// Exit action
//--------------------------------------------------------------------------------------
	IF (me.StateMachine.intState <> me.StateMachine.intStateNext) THEN
		// state is going to change
		;
	END_IF
END_METHOD

{attribute 'object_name' := 'sta_BELTONLYBusy'}
METHOD PROTECTED sta_BELTONLYBusy : BOOL
VAR
	bReady: BOOL;
	iErrorNumber: INT;
END_VAR
// state implemetation

// Entry action
//--------------------------------------------------------------------------------------
	IF (me.StateMachine.intState <> me.StateMachine.intStateLastCycle) THEN
		// state changed since last cycle
		me.StateMachine.intStateLastCycle := me.StateMachine.intState;
		
		// Set Outputs
		p_fbIBH^.setBeltOn();
		p_fbIBH^.setSpeed(In_diSpeed_mm_min := SIf.Par.diSpeed_mm_min);
		THIS^.lastSifPar := SIf.Par;
	END_IF

	
// Cyclic action
//--------------------------------------------------------------------------------------

	// Simulation
	IF (CIf.SwCfg.bolSimulation) THEN
		;
	END_IF
	
	// check if parameters have changed
	IF (TC2_SYSTEM.MEMCMP(pBuf1:=ADR(SIf.Par), pBuf2:=ADR(THIS^.lastSifPar), n:=SIZEOF(SIf.Par)) <> 0) THEN
		p_fbIBH^.setSpeed(In_diSpeed_mm_min := SIf.Par.diSpeed_mm_min);
		THIS^.lastSifPar := SIf.Par;
	END_IF
	
	// check timeouts
	IF me.StateMachine.udiTimeInState_ms>SIf.Par.udiTimeoutBeltOnlyBusy_ms THEN
		iErrorNumber := 100*me.StateMachine.intState+In_iStatus;
		pfbAlarmCtrl^.setAlarm(CIf.Info.intCtrlId,INT_TO_UDINT(E_ALM_OVN.TimeoutError),iErrorNumber,ADR(SIf.Alm),E_AlmState.RST,CIf.Job.eMe_ActivAlmClass);
		me.StateMachine.intStateNext := Base_PLC.cSTA_ERROR;
	ELSIF me.StateMachine.udiTimeInState_ms>SIf.Par.udiTimeoutBeltOnlyReaction_ms THEN
		IF NOT In_bBeltOn OR NOT ((In_iStatus=2) OR (In_iStatus=6)) THEN
			iErrorNumber := 100*me.StateMachine.intState+In_iStatus;
			pfbAlarmCtrl^.setAlarm(CIf.Info.intCtrlId,INT_TO_UDINT(E_ALM_OVN.TimeoutError),iErrorNumber,ADR(SIf.Alm),E_AlmState.RST,CIf.Job.eMe_ActivAlmClass);
			me.StateMachine.intStateNext := Base_PLC.cSTA_ERROR;
		END_IF
	END_IF
	
	// Check if ready
	bReady := TRUE;
	IF NOT In_bBeltOn OR NOT (In_iStatus=2) OR (In_iStatus=6) THEN
		bReady := FALSE;
	END_IF
	IF (ABS(THIS^.In_diSpeed_mm_min - SIf.Par.diSpeed_mm_min) > ABS(SIf.Par.diSpeedBand1_mm_min)) THEN
		bReady := FALSE;
	END_IF
	
	// State Change Condition
	IF (me.StateMachine.intStateNext <> Base_PLC.cSTA_ERROR) THEN
		CASE me.intCmd OF
			// OFF
			Base_PLC.cCMD_OFF:
				me.StateMachine.intStateNext := Base_PLC.cSTA_OFFBusy;
		ELSE
			// DEFAULT
			IF bReady THEN
				me.StateMachine.intStateNext := OVN_CmdState.cSTA_BELTONLY;
			END_IF
		END_CASE
	END_IF


// Exit action
//--------------------------------------------------------------------------------------
	IF (me.StateMachine.intState <> me.StateMachine.intStateNext) THEN
		// state is going to change
		;
	END_IF
END_METHOD

{attribute 'object_name' := 'sta_ERROR'}
METHOD PROTECTED sta_ERROR : BOOL
// state implemetation

// Entry action
//--------------------------------------------------------------------------------------
	IF (me.StateMachine.intState <> me.StateMachine.intStateLastCycle) THEN
		// state changed since last cycle
		me.StateMachine.intStateHistory := me.StateMachine.intStateLastCycle; // -> possibillity to go back to state before error
		me.StateMachine.intStateLastCycle := me.StateMachine.intState;
	END_IF

	
// Cyclic action
//--------------------------------------------------------------------------------------	
	
	// Simulation
	IF (CIf.SwCfg.bolSimulation) THEN
		;
	END_IF
	
	// Mark all tracked item as trash
	fbTracker.markAllTrash();
	
	// auto continue after Connection Error
	IF (iLastCalledAlarmNr=E_ALM_OVN.ConnectionError AND SIf.Cfg.bAutoContinueAfterConnectionError) THEN
		IF THIS^.In_bDriverConnected THEN
			CIf.Job.bolAlmReset := TRUE;
			pfbAlarmCtrl^.setAlarm(CIf.Info.intCtrlId,INT_TO_UDINT(E_ALM_OVN.ConnectionError),UDINT_TO_DINT(THIS^.In_udiDriverErrorID),ADR(SIf.Alm),E_AlmState.CLR,CIf.Job.eMe_ActivAlmClass);
		END_IF
	END_IF
	
	// State Change Condition
	IF (CIf.Job.bolAlmReset = TRUE) THEN
		p_fbIBH^.setAckError();
		me.StateMachine.intStateNext := cSTA_ERRORQuit;
	END_IF


// Exit action
//--------------------------------------------------------------------------------------
	IF (me.StateMachine.intState <> me.StateMachine.intStateNext) THEN
		// state is going to change
		;
	END_IF
END_METHOD

{attribute 'object_name' := 'sta_ERRORQuit'}
METHOD PROTECTED sta_ERRORQuit : BOOL
// state implemetation

// Entry action
//--------------------------------------------------------------------------------------
	IF (me.StateMachine.intState <> me.StateMachine.intStateLastCycle) THEN
		// state changed since last cycle
		me.StateMachine.intStateLastCycle := me.StateMachine.intState;
	END_IF

	
// Cyclic action
//--------------------------------------------------------------------------------------	
	
	// Simulation
	IF (CIf.SwCfg.bolSimulation) THEN
		;
	END_IF
	
	// State Change Condition
	CASE me.StateMachine.intStateHistory OF
		// RUN
		Base_PLC.cSTA_RUN, Base_PLC.cSTA_RUNBusy:
			me.StateMachine.intStateNext := Base_PLC.cSTA_RUNBusy;
		// PON
		Base_PLC.cSTA_PON, Base_PLC.cSTA_PONBusy:
			me.StateMachine.intStateNext := Base_PLC.cSTA_PONBusy;
		// STOP
		Base_PLC.cSTA_STOP, Base_PLC.cSTA_STOPBusy:
			me.StateMachine.intStateNext := Base_PLC.cSTA_STOPBusy;
		// BELTONLY
		OVN_CmdState.cSTA_BELTONLY, OVN_CmdState.cSTA_BELTONLYBusy:
			me.StateMachine.intStateNext := OVN_CmdState.cSTA_BELTONLYBusy;
	ELSE
		// DEFAULT
		me.StateMachine.intStateNext := Base_PLC.cSTA_OFFBusy;
	END_CASE


// Exit action
//--------------------------------------------------------------------------------------
	IF (me.StateMachine.intState <> me.StateMachine.intStateNext) THEN
		// state is going to change
		
		// Reset iLastCalledAlarmNr
		iLastCalledAlarmNr := E_ALM_OVN.NONE;
	END_IF
END_METHOD

{attribute 'object_name' := 'sta_OFF'}
METHOD PROTECTED sta_OFF : BOOL
// state implemetation

// Entry action
//--------------------------------------------------------------------------------------
	IF (me.StateMachine.intState <> me.StateMachine.intStateLastCycle) THEN
		// state changed since last cycle
		me.StateMachine.intStateLastCycle := me.StateMachine.intState;
	END_IF

	
// Cyclic action
//--------------------------------------------------------------------------------------

	// Simulation
	IF (CIf.SwCfg.bolSimulation) THEN
		;
	END_IF
	
	IF NOT In_bOff OR NOT (In_iStatus=1 OR In_iStatus=6 OR In_iStatus=5) THEN
		pfbAlarmCtrl^.setAlarm(CIf.Info.intCtrlId,INT_TO_UDINT(E_ALM_OVN.WrongMode),0,ADR(SIf.Alm),E_AlmState.RST,CIf.Job.eMe_ActivAlmClass);
		me.StateMachine.intStateNext := Base_PLC.cSTA_ERROR;
	END_IF
	
	// State Change Condition
	IF (me.StateMachine.intStateNext <> Base_PLC.cSTA_ERROR) THEN
		CASE me.intCmd OF
			// RUN
			Base_PLC.cCMD_RUN:
				me.StateMachine.intStateNext := Base_PLC.cSTA_RUNBusy;
			// BELTONLY
			OVN_CmdState.cCMD_BELTONLY:
				me.StateMachine.intStateNext := OVN_CmdState.cSTA_BELTONLYBusy;
		ELSE
			// DEFAULT
			;
		END_CASE
	END_IF


// Exit action
//--------------------------------------------------------------------------------------
	IF (me.StateMachine.intState <> me.StateMachine.intStateNext) THEN
		// state is going to change
		;
	END_IF
END_METHOD

{attribute 'object_name' := 'sta_OFFBusy'}
METHOD PROTECTED sta_OFFBusy : BOOL
VAR
	bReady: BOOL;
	iErrorNumber: INT;
END_VAR
// state implemetation

// Entry action
//--------------------------------------------------------------------------------------
	IF (me.StateMachine.intState <> me.StateMachine.intStateLastCycle) THEN
		// state changed since last cycle
		me.StateMachine.intStateLastCycle := me.StateMachine.intState;
		
		// Set Outputs
		p_fbIBH^.setOff();
		
		// mark all tracked items as trash
		fbTracker.markAllTrash();
	END_IF

	
// Cyclic action
//--------------------------------------------------------------------------------------

	// Simulation
	IF (CIf.SwCfg.bolSimulation) THEN
		;
	END_IF
	
	// check timeouts
	IF me.StateMachine.udiTimeInState_ms>SIf.Par.udiTimeoutOffBusy_ms THEN
		iErrorNumber := 100*me.StateMachine.intState+In_iStatus;
		pfbAlarmCtrl^.setAlarm(CIf.Info.intCtrlId,INT_TO_UDINT(E_ALM_OVN.TimeoutError),iErrorNumber,ADR(SIf.Alm),E_AlmState.RST,CIf.Job.eMe_ActivAlmClass);
		me.StateMachine.intStateNext := Base_PLC.cSTA_ERROR;
	ELSIF me.StateMachine.udiTimeInState_ms>SIf.Par.udiTimeoutOffBusyReaction_ms THEN
		IF NOT In_bOff OR NOT ((In_iStatus=1) OR (In_iStatus=6)) THEN
			iErrorNumber := 100*me.StateMachine.intState+In_iStatus;
			pfbAlarmCtrl^.setAlarm(CIf.Info.intCtrlId,INT_TO_UDINT(E_ALM_OVN.TimeoutError),iErrorNumber,ADR(SIf.Alm),E_AlmState.RST,CIf.Job.eMe_ActivAlmClass);
			me.StateMachine.intStateNext := Base_PLC.cSTA_ERROR;
		END_IF
	END_IF
	
	// check if ready
	bReady := TRUE;
	IF NOT In_bOff OR NOT (In_iStatus=1) OR (In_iStatus=6) THEN
		bReady := FALSE;
	END_IF
	
	// State Change Condition
	IF (me.StateMachine.intStateNext <> Base_PLC.cSTA_ERROR) THEN
		IF bReady THEN
			me.StateMachine.intStateNext := Base_PLC.cCMD_OFF;
		END_IF
	END_IF


// Exit action
//--------------------------------------------------------------------------------------
	IF (me.StateMachine.intState <> me.StateMachine.intStateNext) THEN
		// state is going to change
		;
	END_IF
END_METHOD

{attribute 'object_name' := 'sta_PON'}
METHOD PROTECTED sta_PON : BOOL
// state implemetation

// Entry action
//--------------------------------------------------------------------------------------
	IF (me.StateMachine.intState <> me.StateMachine.intStateLastCycle) THEN
		// state changed since last cycle
		me.StateMachine.intStateLastCycle := me.StateMachine.intState;
	END_IF

	
// Cyclic action
//--------------------------------------------------------------------------------------
	
	// Simulation
	IF (CIf.SwCfg.bolSimulation) THEN
		;
	END_IF
	
	// State Change Condition
	IF (me.StateMachine.intStateNext <> Base_PLC.cSTA_ERROR) THEN
		IF me.intCmd>Base_PLC.cCMD_PON THEN
			me.StateMachine.intStateNext := Base_PLC.cSTA_OFFBusy;
		END_IF
	END_IF


// Exit action
//--------------------------------------------------------------------------------------
	IF (me.StateMachine.intState <> me.StateMachine.intStateNext) THEN
		// state is going to change
		;
	END_IF
END_METHOD

{attribute 'object_name' := 'sta_PONBusy'}
METHOD PROTECTED sta_PONBusy : BOOL
VAR
	bReady: BOOL := FALSE;
END_VAR
// state implemetation

// Entry action
//--------------------------------------------------------------------------------------
	IF (me.StateMachine.intState <> me.StateMachine.intStateLastCycle) THEN
		// state changed since last cycle
		me.StateMachine.intStateLastCycle := me.StateMachine.intState;
		
		// Start Driver
		p_fbIBH_CIf^.Job.intACmd := IBH_CmdState.cCMD_CONNECT;
		
		uiNewElementOld_1 := In_uiNewElement_1;
		uiNewElementOld_2 := In_uiNewElement_2;
		uiDeleteElementOld_1 := In_uiDeleteElement_1;
		uiDeleteElementOld_2 := In_uiDeleteElement_2;
	END_IF

	
// Cyclic action
//--------------------------------------------------------------------------------------
	// Simulation
	IF (CIf.SwCfg.bolSimulation) THEN
		;
	END_IF
	
	IF THIS^.In_bDriverError THEN
		pfbAlarmCtrl^.setAlarm(CIf.Info.intCtrlId,INT_TO_UDINT(E_ALM_OVN.ConnectionError),UDINT_TO_DINT(THIS^.In_udiDriverErrorID),ADR(SIf.Alm),E_AlmState.RST,CIf.Job.eMe_ActivAlmClass);
		me.StateMachine.intStateNext := Base_PLC.cSTA_ERROR;
		iLastCalledAlarmNr := E_ALM_OVN.ConnectionError;
	END_IF
	
	// State Change Condition
	IF (me.StateMachine.intStateNext <> Base_PLC.cSTA_ERROR) THEN
		IF (THIS^.In_bDriverConnected) THEN
			me.StateMachine.intStateNext := Base_PLC.cSTA_PON;
		END_IF
	END_IF


// Exit action
//--------------------------------------------------------------------------------------
	IF (me.StateMachine.intState <> me.StateMachine.intStateNext) THEN
		// state is going to change
		;
	END_IF
END_METHOD

{attribute 'object_name' := 'sta_RUN'}
METHOD PROTECTED sta_RUN : BOOL
VAR
	uiIdx: UINT;
	bOutOfBand: BOOL := FALSE;
	bError: BOOL := FALSE;
END_VAR
// state implemetation

// Entry action
//--------------------------------------------------------------------------------------
	IF (me.StateMachine.intState <> me.StateMachine.intStateLastCycle) THEN
		// state changed since last cycle
		me.StateMachine.intStateLastCycle := me.StateMachine.intState;
		THIS^.lastSifPar := SIf.Par;
		
		// reset monitor timeouts
		fbSpeedMonitor.resetTime();
		FOR uiIdx:=0 TO SIf.Cfg.uiNumberOfModules-1 BY 1 DO
			afbTempMonitors[uiIdx].resetTime();
			afbAirMonitors[uiIdx].resetTime();
		END_FOR
	END_IF

	
// Cyclic action
//--------------------------------------------------------------------------------------

	// Simulation
	IF (CIf.SwCfg.bolSimulation) THEN
		;
	END_IF
	
	// check if parameters have changed
	IF (TC2_SYSTEM.MEMCMP(pBuf1:=ADR(SIf.Par), pBuf2:=ADR(THIS^.lastSifPar), n:=SIZEOF(SIf.Par)) <> 0) THEN
		me.StateMachine.intStateNext := Base_PLC.cSTA_RUNBusy;
	END_IF
	
	IF NOT In_bRun OR NOT (In_iStatus=4 OR In_iStatus=6 OR In_iStatus=5) THEN
		pfbAlarmCtrl^.setAlarm(CIf.Info.intCtrlId,INT_TO_UDINT(E_ALM_OVN.WrongMode),0,ADR(SIf.Alm),E_AlmState.RST,CIf.Job.eMe_ActivAlmClass);
		me.StateMachine.intStateNext := Base_PLC.cSTA_ERROR;
	END_IF
	
	// Update Monitors
	IF (me.StateMachine.intStateNext <> Base_PLC.cSTA_RUNBusy) THEN
		// temperature monitors
		FOR uiIdx:=0 TO SIf.Cfg.uiNumberOfModules-1 BY 1 DO
			afbTempMonitors[uiIdx](	diCurrentValue		:= THIS^.SIf.Cur.adiTemp_dc[uiIdx],
									diTargetValue		:= THIS^.SIf.Par.adiTemp_dc[uiIdx],
									diBand1				:= THIS^.SIf.Par.adiTempBand1_dc[uiIdx],
									diBand2				:= THIS^.SIf.Par.adiTempBand2_dc[uiIdx],
									udiTimeout_ms		:= THIS^.SIf.Par.audiTempTimeout_ms[uiIdx],
									udiSampleTime_ms	:= me.FUBInfo.udiSample_ms,
									bOutOfBand			=> bOutOfBand,
									bError				=> bError);
			IF (bError = TRUE) THEN
				pfbAlarmCtrl^.setAlarm(CIf.Info.intCtrlId,INT_TO_UDINT(E_ALM_OVN.TempError),uiIdx,ADR(SIf.Alm),E_AlmState.RST,CIf.Job.eMe_ActivAlmClass);
				me.StateMachine.intStateNext := Base_PLC.cSTA_ERROR;
			END_IF
		END_FOR
		// airflow monitors
		FOR uiIdx:=0 TO SIf.Cfg.uiNumberOfModules-1 BY 1 DO
			afbAirMonitors[uiIdx](	diCurrentValue		:= THIS^.SIf.Cur.adiAir_p[uiIdx],
									diTargetValue		:= THIS^.SIf.Par.adiAir_p[uiIdx],
									diBand1				:= THIS^.SIf.Par.adiAirBand1_p[uiIdx],
									diBand2				:= THIS^.SIf.Par.adiAirBand2_p[uiIdx],
									udiTimeout_ms		:= THIS^.SIf.Par.audiAirTimeout_ms[uiIdx],
									udiSampleTime_ms	:= me.FUBInfo.udiSample_ms,
									bOutOfBand			=> bOutOfBand,
									bError				=> bError);
			IF (bError = TRUE) THEN
				pfbAlarmCtrl^.setAlarm(CIf.Info.intCtrlId,INT_TO_UDINT(E_ALM_OVN.AirError),uiIdx,ADR(SIf.Alm),E_AlmState.RST,CIf.Job.eMe_ActivAlmClass);
				me.StateMachine.intStateNext := Base_PLC.cSTA_ERROR;
			END_IF
		END_FOR
		// band speed monitor
		fbSpeedMonitor(	diCurrentValue		:= THIS^.SIf.Cur.diSpeed_mm_min,
						diTargetValue		:= THIS^.SIf.Par.diSpeed_mm_min,
						diBand1				:= THIS^.SIf.Par.diSpeedBand1_mm_min,
						diBand2				:= THIS^.SIf.Par.diSpeedBand2_mm_min,
						udiTimeout_ms		:= THIS^.SIf.Par.udiSpeedTimeout_ms,
						udiSampleTime_ms	:= me.FUBInfo.udiSample_ms,
						bOutOfBand			=> bOutOfBand,
						bError				=> bError);
		IF (bError = TRUE) THEN
			pfbAlarmCtrl^.setAlarm(CIf.Info.intCtrlId,INT_TO_UDINT(E_ALM_OVN.SpeedError),0,ADR(SIf.Alm),E_AlmState.RST,CIf.Job.eMe_ActivAlmClass);
			me.StateMachine.intStateNext := Base_PLC.cSTA_ERROR;
		END_IF
	END_IF
	
	// State Change Condition
	IF (me.StateMachine.intStateNext <> Base_PLC.cSTA_ERROR) THEN
		CASE me.intCmd OF
			// OFF
			Base_PLC.cCMD_OFF:
				me.StateMachine.intStateNext := Base_PLC.cSTA_OFFBusy;
			// BELTONLY
			OVN_CmdState.cCMD_BELTONLY:
				me.StateMachine.intStateNext := Base_PLC.cSTA_OFFBusy;
		ELSE
			// DEFAULT
			;
		END_CASE
	END_IF


// Exit action
//--------------------------------------------------------------------------------------
	IF (me.StateMachine.intState <> me.StateMachine.intStateNext) THEN
		// state is going to change
		;
	END_IF
END_METHOD

{attribute 'object_name' := 'sta_RUNBusy'}
METHOD PROTECTED sta_RUNBusy : BOOL
VAR
	iIdx: UINT;
	bReady: BOOL;
	iErrorNumber: INT;
END_VAR
// state implemetation

// Entry action
//--------------------------------------------------------------------------------------
	IF (me.StateMachine.intState <> me.StateMachine.intStateLastCycle) THEN
		// state changed since last cycle
		me.StateMachine.intStateLastCycle := me.StateMachine.intState;
		
		// Set Outputs
		p_fbIBH^.setRun();
		p_fbIBH^.setSpeed(In_diSpeed_mm_min := SIf.Par.diSpeed_mm_min);
		p_fbIBH^.setTemp(In_adiTemp_dc := SIf.Par.adiTemp_dc);
		p_fbIBH^.setAirflow(In_adiAir_p := SIf.Par.adiAir_p);
		THIS^.lastSifPar := SIf.Par;
		
		udiTimeInBand := 0;
		
		// delete all tracked items
		fbTracker.deleteAll();
	END_IF
	
// Cyclic action
//--------------------------------------------------------------------------------------

	// Simulation 
	IF (CIf.SwCfg.bolSimulation) THEN
		;
	END_IF
	
	// check if parameters have changed
	IF (TC2_SYSTEM.MEMCMP(pBuf1:=ADR(SIf.Par), pBuf2:=ADR(THIS^.lastSifPar), n:=SIZEOF(SIf.Par)) <> 0) THEN
		p_fbIBH^.setSpeed(In_diSpeed_mm_min := SIf.Par.diSpeed_mm_min);
		p_fbIBH^.setTemp(In_adiTemp_dc := SIf.Par.adiTemp_dc);
		p_fbIBH^.setAirflow(In_adiAir_p := SIf.Par.adiAir_p);
		THIS^.lastSifPar := SIf.Par;
	END_IF
	
	// check timeouts
	IF me.StateMachine.udiTimeInState_ms>SIf.Par.udiTimeoutRunBusyReaction_ms THEN
		IF NOT In_bRun OR NOT ((In_iStatus=0) OR (In_iStatus=4) OR (In_iStatus=6)) THEN
			iErrorNumber := 100*me.StateMachine.intState+In_iStatus;
			pfbAlarmCtrl^.setAlarm(CIf.Info.intCtrlId,INT_TO_UDINT(E_ALM_OVN.TimeoutError),iErrorNumber,ADR(SIf.Alm),E_AlmState.RST,CIf.Job.eMe_ActivAlmClass);
			me.StateMachine.intStateNext := Base_PLC.cSTA_ERROR;
		END_IF
	END_IF
	
	// Check if ready
	bReady := TRUE;
	IF NOT In_bRun OR NOT (In_iStatus=4) OR (In_iStatus=6) THEN
		bReady := FALSE;
	END_IF
	IF (ABS(THIS^.In_diSpeed_mm_min - SIf.Par.diSpeed_mm_min) > ABS(SIf.Par.diSpeedBand1_mm_min)) THEN
		bReady := FALSE;
	END_IF
	FOR iIdx:=0 TO SIf.Cfg.uiNumberOfModules-1 BY 1 DO
		// Temperature
		IF (ABS(THIS^.In_adiTemp_dc[iIdx] - SIf.Par.adiTemp_dc[iIdx]) > ABS(THIS^.SIf.Par.adiTempBand1_dc[iIdx])) THEN
			bReady := FALSE;
		END_IF
		// Airflow
		IF (ABS(THIS^.In_adiAir_p[iIdx] - THIS^.SIf.Par.adiAir_p[iIdx]) > ABS(THIS^.SIf.Par.adiAirBand1_p[iIdx])) THEN
			bReady := FALSE;
		END_IF
	END_FOR
	
	IF bReady THEN
		udiTimeInBand := udiTimeInBand + me.FUBInfo.udiSample_ms;
		IF udiTimeInBand < SIf.Par.udiTimeoutRunBusyInBand_ms THEN
			bReady := FALSE;
		END_IF
	ELSE
		udiTimeInBand := 0;
	END_IF
	
	// State Change Condition
	IF (me.StateMachine.intStateNext <> Base_PLC.cSTA_ERROR) THEN
		CASE me.intCmd OF
			// OFF
			Base_PLC.cCMD_OFF:
				me.StateMachine.intStateNext := Base_PLC.cSTA_OFFBusy;
			// BELTONLY
			OVN_CmdState.cCMD_BELTONLY:
				me.StateMachine.intStateNext := Base_PLC.cSTA_OFFBusy;
		ELSE
			// DEFAULT
			IF bReady THEN
				me.StateMachine.intStateNext := Base_PLC.cSTA_RUN;
			END_IF
		END_CASE
	END_IF

		
// Exit action
//--------------------------------------------------------------------------------------
	IF (me.StateMachine.intState <> me.StateMachine.intStateNext) THEN
		// state is going to change
		;
	END_IF
END_METHOD

{attribute 'object_name' := 'StateMachine'}
METHOD PROTECTED StateMachine : BOOL
SUPER^.StateMachine();

// main statemachine of base controller
CASE me.StateMachine.intState OF
	// BELTONLY
    OVN_CmdState.cSTA_BELTONLY: 
        THIS^.sta_BELTONLY();
    OVN_CmdState.cSTA_BELTONLYBusy: 
        THIS^.sta_BELTONLYBusy();
	// RUN
	Base_PLC.cSTA_RUN:
		THIS^.sta_RUN();
	Base_PLC.cSTA_RUNBusy:
		THIS^.sta_RUNBusy();
END_CASE;
END_METHOD

END_FUNCTION_BLOCK

// POUs/Controller/Lvl1/OVN (Oven)/FB_Tracker
FUNCTION_BLOCK FB_Tracker
VAR
	fbList: FB_DLL(In_bDoDataWipe := FALSE);
	udiSampleTime_us: UDINT;
	uiNumberOfModules: UINT;
	diModuleLength_mm: DINT;
	diDistanceBeforeOven_mm: DINT;
	diDistanceAfterOven_mm: DINT;
	pDataChannelFifo: POINTER TO FB_DataChannelSenderFifo;
END_VAR

{attribute 'object_name' := 'addElement'}
METHOD addElement
VAR_INPUT
	In_uliBarcode: ULINT;
END_VAR
VAR
	pData: POINTER TO T_Data;
	uiIdx: UINT;
END_VAR
pData := __NEW(T_Data);
pData^.uliBarcode := In_uliBarcode;
pData^.bTrash := FALSE;
pData^.bBarcodeMissed := FALSE;
pData^.diDistance_um := 0;
FOR uiIdx:=0 TO MAX_NUMBER_OF_OVEN_MODULES-1 BY 1 DO
	pData^.diCyclesInModule[uiIdx] := 0;
	pData^.diSumTemp_mc[uiIdx] := 0;
END_FOR

fbList.addElement(In_uliKey:=In_uliBarcode, In_pData:=pData);
END_METHOD

PROPERTY DataChannel : POINTER TO FB_DataChannelSenderFifo
SET
pDataChannelFifo := DataChannel;
END_SET
END_PROPERTY

{attribute 'object_name' := 'deleteAll'}
METHOD deleteAll
fbList.deleteAll();
END_METHOD

{attribute 'object_name' := 'deleteElement'}
METHOD deleteElement : BOOL
VAR_INPUT
	uliBarcodeOfElement: ULINT;
	bolSendToSaber: BOOL;
END_VAR
VAR
	pDeleteElement: POINTER TO T_Element;
	pData: POINTER TO T_Data;
END_VAR
pDeleteElement := fbList.searchElement(In_uliKey:=uliBarcodeOfElement);

IF (pDeleteElement <> 0) THEN
	
	deleteElement := TRUE;
	pData := fbList.deleteElement(pDeleteElement);

	IF bolSendToSaber THEN
		sendData(pData);
	END_IF

	__DELETE(pData);
ELSE
	deleteElement := FALSE;
END_IF
END_METHOD

PROPERTY distanceAfterOven_mm : DINT
GET
distanceAfterOven_mm := diDistanceAfterOven_mm;
END_GET
SET
diDistanceAfterOven_mm := distanceAfterOven_mm;
END_SET
END_PROPERTY

PROPERTY distanceBeforeOven_mm : DINT
GET
distanceBeforeOven_mm := diDistanceBeforeOven_mm;
END_GET
SET
diDistanceBeforeOven_mm := distanceBeforeOven_mm;
END_SET
END_PROPERTY

{attribute 'object_name' := 'markAllTrash'}
METHOD markAllTrash
VAR
	pCurrentElement: POINTER TO T_Element;
	pCurrentData: POINTER TO T_Data;
	uiIdx: UINT;
END_VAR
pCurrentElement := fbList.firstElement();

WHILE (pCurrentElement <> 0) DO
	pCurrentData := pCurrentElement^.pData;
	pCurrentData^.bTrash := TRUE;
	pCurrentElement := pCurrentElement^.pNextElement;
END_WHILE
END_METHOD

PROPERTY moduleLength_mm : DINT
GET
moduleLength_mm := diModuleLength_mm;
END_GET
SET
diModuleLength_mm := moduleLength_mm;
END_SET
END_PROPERTY

{attribute 'object_name' := 'numberOfElements'}
METHOD numberOfElements : UINT
numberOfElements := fbList.numberOfElements();
END_METHOD

PROPERTY numberOfModules : UINT
GET
numberOfModules := uiNumberOfModules;
END_GET
SET
uiNumberOfModules := numberOfModules;
END_SET
END_PROPERTY

PROPERTY sampleTime_us : UDINT
GET
sampleTime_us := udiSampleTime_us;
END_GET
SET
udiSampleTime_us := sampleTime_us;
END_SET
END_PROPERTY

{attribute 'object_name' := 'sendData'}
METHOD sendData : BOOL
VAR_INPUT
	pData: POINTER TO T_Data;
END_VAR
VAR
	uiIdx: UINT;
	pItem: POINTER TO T_Oven_DCH;
END_VAR
IF pDataChannelFifo <> NULL THEN
	pItem := __NEW(T_Oven_DCH);

	// prepare temperature values
	FOR uiIdx:=0 TO MAX_NUMBER_OF_OVEN_MODULES-1 BY 1 DO
		IF pData^.diCyclesInModule[uiIdx] > 0 THEN
			pItem^.diTemperature_mc[uiIdx] := pData^.diSumTemp_mc[uiIdx]/pData^.diCyclesInModule[uiIdx];
		ELSE
			pItem^.diTemperature_mc[uiIdx] := 0;
		END_IF
	END_FOR

	pItem^.rBaseInfo.bolItemAvailable := TRUE;
	
	IF pData^.bTrash THEN
		pItem^.rBaseInfo.eHealth := E_ItemHealth.Ovn_Temperature;
	ELSE
		pItem^.rBaseInfo.eHealth := E_ItemHealth.Healthy;
	END_IF
	pItem^.bTrash := pData^.bTrash;
	
	pItem^.udiIdentification := pData^.uliBarcode;

	pDataChannelFifo^.Push(pItem);
END_IF
END_METHOD

{attribute 'object_name' := 'update'}
METHOD update
VAR_INPUT
	In_adiTemp_mc: ARRAY[0..(MAX_NUMBER_OF_OVEN_MODULES - 1)] OF DINT;
	In_diSpeed_mm_min: DINT;
	bolSendToSaber: BOOL;
END_VAR
VAR
	pCurrentElement: POINTER TO T_Element;
	pCurrentData: POINTER TO T_Data;
	uiIdx: UINT;
END_VAR
pCurrentElement := fbList.firstElement();

WHILE (pCurrentElement <> 0) DO
	pCurrentData := pCurrentElement^.pData;
	
	// Distance
	pCurrentData^.diDistance_um := pCurrentData^.diDistance_um + In_diSpeed_mm_min*1000/60/1000000*UDINT_TO_DINT(udiSampleTime_us);
	
	IF ( pCurrentData^.diDistance_um < (diDistanceBeforeOven_mm * 1000) ) THEN
		// Before the Oven
		;
	ELSIF (pCurrentData^.diDistance_um > (diDistanceBeforeOven_mm+diDistanceAfterOven_mm+uiNumberOfModules*diModuleLength_mm+1000)*1000) THEN
		// 1m after the Barcode scanners after the Oven
		pCurrentData^.bBarcodeMissed := TRUE;
		deleteElement(uliBarcodeOfElement:=pCurrentData^.uliBarcode,bolSendToSaber:=bolSendToSaber);
	ELSE
		// In the Oven
		FOR uiIdx:=0 TO uiNumberOfModules-1 BY 1 DO
			IF (	(pCurrentData^.diDistance_um >= (diDistanceBeforeOven_mm + uiIdx*diModuleLength_mm)*1000)
				AND (pCurrentData^.diDistance_um < (diDistanceBeforeOven_mm + (uiIdx+1)*diModuleLength_mm)*1000) ) THEN
				pCurrentData^.diCyclesInModule[uiIdx] := pCurrentData^.diCyclesInModule[uiIdx] + 1;
				pCurrentData^.diSumTemp_mc[uiIdx] := pCurrentData^.diSumTemp_mc[uiIdx] + In_adiTemp_mc[uiIdx];
			END_IF
		END_FOR
	END_IF
	
	pCurrentElement := pCurrentElement^.pNextElement;
END_WHILE
END_METHOD

END_FUNCTION_BLOCK

// POUs/Controller/Lvl1/PTA [Paper Transport Alignment]/helper/cycle_Pta
FUNCTION cycle_Pta : BOOL
VAR_INPUT
	pPta: POINTER TO T_PTA;
END_VAR

pPta^.ctrl.fbPta_Umc.In_bolEmoOk				:= pPta^.io.In_bolUmc_EmoOk;
pPta^.ctrl.fbPta_Umc.In_uinStatus 				:= pPta^.io.In_uinUmc_Status;
pPta^.ctrl.fbPta_Umc.In_intMotorActualSpeed 	:= pPta^.io.In_uinUmc_ActualSpeed;
pPta^.ctrl.fbPta_Umc.In_uinMotorSetSpeed 		:= pPta^.io.In_uinUmc_SetSpeed;
pPta^.ctrl.fbPta_Umc.In_uinECATState 			:= pPta^.io.In_uinUmc_ECatState;
pPta^.ctrl.fbPta_Umc.In_strNetId 				:= pPta^.io.In_strUmc_ECatNetId;
pPta^.ctrl.fbPta_Umc.In_uintPort 				:= pPta^.io.In_uinUmc_ECatPort;
pPta^.ctrl.fbPta_Umc();
pPta^.io.Out_uinUmc_SetSpeed 					:= pPta^.ctrl.fbPta_Umc.Out_uinSpeedSetpoint;
pPta^.io.Out_uinUmc_Control 					:= pPta^.ctrl.fbPta_Umc.Out_uinControl;

pPta^.ctrl.fbPta.In_bolBeltEntrySensor		 	:= pPta^.io.In_bolInputSensor;
pPta^.ctrl.fbPta.In_bolBeltExitSensor 			:= pPta^.io.In_bolOutputSensor;
pPta^.ctrl.fbPta();

END_FUNCTION

// POUs/Controller/Lvl1/PTA [Paper Transport Alignment]/helper/init_Pta
FUNCTION init_Pta : BOOL
VAR_INPUT
	pPta			: POINTER TO T_PTA;
	/// instance array of all controller instances
	pCtrlInst		: POINTER TO fb_CtrlBase;
	/// common interface array of all controllers (main use for PLC)
	pCtrlCIf		: POINTER TO T_Ctrl_CIf;
END_VAR

pPta^.ctrl.fbPta_Umc.iniAllCtrlArrays(pCtrlInst,pCtrlCIf,pPta^.id.Pta_Umc);
pPta^.ctrl.fbPta.iniAllCtrlArrays(pCtrlInst,pCtrlCIf,pPta^.id.Pta);
pPta^.ctrl.fbPta.Drive := ADR(pPta^.ctrl.fbPta_Umc);

// PTA is a special type of PTB
pPta^.ctrl.fbPta.CtrlSIf^.Cfg.bolVacuumPresent := FALSE;

END_FUNCTION

// POUs/Controller/Lvl1/PTB [Paper Transport Belt]/helper/cycle_Ptb
FUNCTION cycle_Ptb : BOOL
VAR_INPUT
	pPtb: POINTER TO T_PTB;
END_VAR

pPtb^.ctrl.fbPtb_Umc.In_bolEmoOk				:= pPtb^.io.In_bolUmc_EmoOk;
pPtb^.ctrl.fbPtb_Umc.In_uinStatus 				:= pPtb^.io.In_uinUmc_Status;
pPtb^.ctrl.fbPtb_Umc.In_intMotorActualSpeed 	:= pPtb^.io.In_uinUmc_ActualSpeed;
pPtb^.ctrl.fbPtb_Umc.In_uinMotorSetSpeed 		:= pPtb^.io.In_uinUmc_SetSpeed;
pPtb^.ctrl.fbPtb_Umc.In_uinECATState 			:= pPtb^.io.In_uinUmc_ECatState;
pPtb^.ctrl.fbPtb_Umc.In_strNetId 				:= pPtb^.io.In_strUmc_ECatNetId;
pPtb^.ctrl.fbPtb_Umc.In_uintPort 				:= pPtb^.io.In_uinUmc_ECatPort;
pPtb^.ctrl.fbPtb_Umc();
pPtb^.io.Out_uinUmc_SetSpeed 					:= pPtb^.ctrl.fbPtb_Umc.Out_uinSpeedSetpoint;
pPtb^.io.Out_uinUmc_Control 					:= pPtb^.ctrl.fbPtb_Umc.Out_uinControl;

pPtb^.ctrl.fbPtb_Vpc.In_bolPumpOk 				:= pPtb^.io.In_bolVpc_PumpOk;
pPtb^.ctrl.fbPtb_Vpc.In_bolVacuumOk 			:= pPtb^.io.In_bolVpc_VacuumSensor;
pPtb^.ctrl.fbPtb_Vpc();
pPtb^.io.Out_bolVpc_PumpOn 						:= pPtb^.ctrl.fbPtb_Vpc.Out_bolVaccumPumpOn;

pPtb^.ctrl.fbPtb.In_bolBeltEntrySensor		 	:= pPtb^.io.In_bolInputSensor;
pPtb^.ctrl.fbPtb.In_bolBeltExitSensor 			:= pPtb^.io.In_bolOutputSensor;
pPtb^.ctrl.fbPtb();

END_FUNCTION

// POUs/Controller/Lvl1/PTB [Paper Transport Belt]/helper/init_Ptb
FUNCTION init_Ptb : BOOL
VAR_INPUT
	pPtb			: POINTER TO T_PTB;
	/// instance array of all controller instances
	pCtrlInst		: POINTER TO fb_CtrlBase;
	/// common interface array of all controllers (main use for PLC)
	pCtrlCIf		: POINTER TO T_Ctrl_CIf;
END_VAR

pPtb^.ctrl.fbPtb_Vpc.iniAllCtrlArrays(pCtrlInst,pCtrlCIf,pPtb^.id.Ptb_Vpc);
pPtb^.ctrl.fbPtb_Umc.iniAllCtrlArrays(pCtrlInst,pCtrlCIf,pPtb^.id.Ptb_Umc);
pPtb^.ctrl.fbPtb.iniAllCtrlArrays(pCtrlInst,pCtrlCIf,pPtb^.id.Ptb);
pPtb^.ctrl.fbPtb.Drive := ADR(pPtb^.ctrl.fbPtb_Umc);
pPtb^.ctrl.fbPtb.VacuumPump := ADR(pPtb^.ctrl.fbPtb_Vpc);

END_FUNCTION

// POUs/Controller/Lvl1/PTB [Paper Transport Belt]/FB_PTB
FUNCTION_BLOCK FB_PTB EXTENDS FB_CtrlBase
VAR_INPUT
	In_bolBeltEntrySensor		: BOOL;
	In_bolBeltExitSensor		: BOOL;
END_VAR
VAR_OUTPUT
END_VAR
VAR
	/// Specific interface struct for public access
	SIf					: T_Ctrl_SIf_PTB;
	///pointer to function block
	p_fbMotor				: POINTER TO FB_UMC;
	pMotorCIf				: POINTER TO T_Ctrl_CIf;
	p_fbPump				: POINTER TO FB_VPC;
	pPumpCIf				: POINTER TO T_Ctrl_CIf;
	fbEntrySensorDebounce	: FB_PRS;
	fbExitSensorDebounce	: FB_PRS;
	arMotorDirection		: ARRAY [0..E_BELT_DIRECTION.MAX_E_BELT_DIRECTION-1] OF E_TURN_DIRECTION;
	
	// Paper Position Service
	fbPositionService		: FB_PTR;
	udiIdCounter			: UDINT;
	
	// Paper Edge Detectors
	fbPaperEntryPEdge					: TC2_STANDARD.R_TRIG;
	fbPaperEntryNEdge					: TC2_STANDARD.F_TRIG;
	fbPaperExitPEdge					: TC2_STANDARD.R_TRIG;
	fbPaperExitNEdge					: TC2_STANDARD.F_TRIG;
	
END_VAR

(*__________________________________________________________________________________________________
¦	
¦	Vistaprint Schweiz GmbH
¦	CH - 8401 Winterthur
¦
¦	www.vistaprint.ch - info@vistaprint.ch
¦___________________________________________________________________________________________________

Function desription:
Vacuum Pump implementation. 


History:
Version		Date			Author		Comment
---------------------------------------------------------------------------------------------------
0.00.1		09.07.2013		PC			Start history
0.00.2		14.02.2014		AVME/MRU	Cyclic call of fbPositionService added
0.00.3		24.02.2014		AVME/MRU	sta_OFFBusy reworked
0.00.4		02.10.2014		AVME/MRU	Alwaysw reworked for Single_Answer
___________________________________________________________________________________________________*)


SUPER^();

(*
IF (me.bolActivate) THEN // cyclic call enabled
	IF (CIf.Info.bolInitDone=FALSE) THEN // first cycle -> init
		CtrlInit();
		CIf.Info.bolInitDone := TRUE;
	ELSE
		CycleStartDuty();
	
		Always();
		
		StateMachine();
		
		CycleEndDuty();
	END_IF
END_IF;
*)

METHOD PROTECTED Always : BOOL
SUPER^.Always();

// ----------------------------------------------------------------------------------
// cyclic actions outside of statemachine
IF (me.StateMachine.intState<>cSTA_SINGLE_ANSWER) THEN
	
	; // always error supervision
	
END_IF

// ----------------------------------------------------------------------------------
// Conditions Always
IF (((me.Alarm.eActivAlmClass=E_AlmClass.EOFF) OR (me.Alarm.eActivAlmClass=E_AlmClass.OFF) OR (me.intCmd=cCMD_OFF))
		 AND (me.StateMachine.intState<>cSTA_ERROR) AND (me.StateMachine.intState<>cSTA_ERRORQuit) AND
		(me.StateMachine.intState<>cSTA_OFF) AND (me.StateMachine.intState<>cSTA_OFFBusy) AND (me.StateMachine.intState<>cSTA_SINGLE_ANSWER)) THEN
	// alarm evt EOFF, OFF or cmd off
	me.StateMachine.intStateNext := cSTA_OFFBusy;
END_IF

// ----------------------------------------------------------------------------------
// Conditions Always
// overrule error always from base -> no EOFF State!! in EOFF go to OFF
IF (me.StateMachine.intStateNext = cSTA_EOFFBusy) THEN
	IF (me.StateMachine.intState=cSTA_OFF) THEN
		me.StateMachine.intStateNext := cSTA_OFF;
	ELSE // stay in OFF
		me.StateMachine.intStateNext := cSTA_OFFBusy;
	END_IF
END_IF

// -----------------------------------------------------------------------------------
PaperPositionHandling();
// -----------------------------------------------------------------------------------
END_METHOD

METHOD PROTECTED CalculateBeltParameter : UINT
VAR_INPUT
	uinBeltSpeed_mms		: UINT;   	// Belt speed in mm/sec
	reaRpmDistance			: REAL;		// mm/rotation
	pCur		: POINTER TO T_Belt_Cur_Base;
END_VAR
pCur^.uinBeltSpeed_mms := uinBeltSpeed_mms;
// RPM = Speed [mm/sec] / Dispance per Rotation [mm/rpm]
pCur^.uinBeltSpeed_rpm := REAL_TO_UINT(UINT_TO_REAL(uinBeltSpeed_mms) * 60.0 / reaRpmDistance);

CalculateBeltParameter := pCur^.uinBeltSpeed_rpm;
END_METHOD

METHOD PROTECTED CalculateModeParameter : BOOL
VAR_INPUT
END_VAR
CASE SIf.Cfg.eMode OF  
	E_PTB_MODE.ToDistance:
		SIf.Cur.udiTimeToMove_ms		:= REAL_TO_UDINT( 1000.0 * UDINT_TO_REAL(SIf.Par.udiDistanceToMove_mm) / UINT_TO_REAL(SIf.Par.rBeltParam.uinBeltSpeed));
		SIf.Cur.udiTimeToMove_ms		:= SIf.Cur.udiTimeToMove_ms + p_fbMotor^.CtrlSIf^.Par.udiMoveStartLatency - p_fbMotor^.CtrlSIf^.Par.udiMoveStopLatency;
		SIf.Cur.udiDistanceToMove_mm	:= SIf.Par.udiDistanceToMove_mm;
	E_PTB_MODE.ToTime:
		SIf.Cur.udiTimeToMove_ms		:= SIf.Par.udiTimeToMove_ms;
		SIf.Cur.udiDistanceToMove_mm	:= SIf.Par.udiTimeToMove_ms * UINT_TO_UDINT(SIf.Par.rBeltParam.uinBeltSpeed) / 1000;
		SIf.Cur.udiTimeToMove_ms		:= SIf.Cur.udiTimeToMove_ms + p_fbMotor^.CtrlSIf^.Par.udiMoveStartLatency - p_fbMotor^.CtrlSIf^.Par.udiMoveStopLatency;
ELSE
	SIf.Cur.udiTimeToMove_ms		:= 0;
	SIf.Cur.udiDistanceToMove_mm	:= 0;
END_CASE
END_METHOD

METHOD PROTECTED CheckPumpState : BOOL
VAR_INPUT
	intState		: INT;
END_VAR
CheckPumpState := TRUE;

IF SIf.Cfg.bolVacuumPresent THEN
	CheckPumpState := p_fbPump^.CtrlCIf^.Job.intState = intState;
END_IF
END_METHOD

ACTION cmd_OFF:
p_fbMotor^.CtrlCIf^.Job.intACmd := BASE_PLC.cCMD_OFF;
SetPumpComand(cCMD_OFF);
END_ACTION

METHOD PROTECTED cmd_RUN : BOOL
VAR_INPUT
	uinBeltSpeed			: UINT;
END_VAR
SIf.Cur.eActualDirection := SIf.Par.intDirection;
SIf.Cur.rBeltParam.uinBeltSpeed_rpm := CalculateBeltParameter(
											uinBeltSpeed,
											sif.Cfg.rBeltParam.reaRpmDistance_mm,
											ADR(SIf.Cur.rBeltParam));
CalculateModeParameter();
p_fbMotor^.CtrlSIf^.Par.eRotationDirection 	:= THIS^.arMotorDirection[SIf.Par.intDirection];
p_fbMotor^.CtrlSIf^.Par.uinSpeed_rpm 		:= SIf.Cur.rBeltParam.uinBeltSpeed_rpm;
p_fbMotor^.CtrlCIf^.Job.intACmd :=BASE_PLC.cCMD_RUN;
SetPumpComand(cCMD_RUN);
END_METHOD

ACTION cmd_STOP:
p_fbMotor^.CtrlCIf^.Job.intACmd := BASE_PLC.cCMD_STOP;
SetPumpComand(cCMD_RUN);
END_ACTION

METHOD PUBLIC CtrlInit : BOOL
VAR_INPUT
END_VAR
SUPER^.CtrlInit();

pMotorCIf := p_fbMotor^.CtrlCIf;
AddChild(p_fbMotor^);

IF SIf.Cfg.bolVacuumPresent THEN
	pPumpCIf  := p_fbPump^.CtrlCIf;
	AddChild(p_fbPump^);
END_IF

arMotorDirection[E_BELT_DIRECTION.BACKWARD] := SIf.Cfg.rBeltParam.intBackwardDirection;
arMotorDirection[E_BELT_DIRECTION.FORWARD] := SIf.Cfg.rBeltParam.intForwardDirection;

fbPositionService.TimeBase := me.FUBInfo.udiSample_us;
fbPositionService.BeltLength := UDINT_TO_DINT(SIf.Par.udiBeltLength_mm);

CASE SIf.Par.ePaperOrientation OF
	E_PTB_PaperDirection.Portrait:
		fbPositionService.PaperEntryOffset := UINT_TO_INT(SIf.Par.uinPaperHight_mm); 
	E_PTB_PaperDirection.Landscape:
		fbPositionService.PaperEntryOffset := UINT_TO_INT(SIf.Par.uinPaperWidth_mm); 
END_CASE

SIf.Cur.pPositionList := fbPositionService.PositionList;
udiIdCounter := 0;
END_METHOD

PROPERTY PUBLIC CtrlSIf : POINTER TO T_Ctrl_SIf_PTB
GET
CtrlSIf := ADR(SIf);
END_GET
SET
END_SET
END_PROPERTY

PROPERTY PUBLIC Drive :  POINTER TO FB_UMC
GET
Drive := p_fbMotor;
END_GET
SET
p_fbMotor := Drive;
END_SET
END_PROPERTY

METHOD FB_init : BOOL
VAR_INPUT
	bInitRetains : BOOL; // if TRUE, the retain variables are initialized (warm start / cold start)
	bInCopyCode : BOOL;  // if TRUE, the instance afterwards gets moved into the copy code (online change)
END_VAR
VAR
	iIdx		: UINT;
	iLength		: UINT;	
END_VAR
//------------------------------------------------------------------------------------------------------------------------
// to manually change in new FUB implementation!!!
// define valid commands for this controller
iLength := SIZEOF(CIf.Job.aCmdList)/SIZEOF(CIf.Job.aCmdList[0]);
iIdx := 0;

WHILE (iIdx < iLength) AND (CIf.Job.aCmdList[iIdx].intCmd <> cCMD_INITIALIZED) DO
	iIdx := iIdx + 1; 
END_WHILE

IF (iIdx < iLength) THEN
// Add configuration of own comands	
	CIf.Job.aCmdList[iIdx].intCmd := BASE_PLC.cCMD_RUN;
	CIf.Job.aCmdList[iIdx].strName := 'Run'; 
	CIf.Job.aCmdList[iIdx].bolAvailable := TRUE;
	iIdx := iIdx + 1;
	CIf.Job.aCmdList[iIdx].intCmd := BASE_PLC.cCMD_STOP;
	CIf.Job.aCmdList[iIdx].strName := 'Stop'; 
	CIf.Job.aCmdList[iIdx].bolAvailable := TRUE;
	iIdx := iIdx + 1;
	CIf.Job.aCmdList[iIdx].intCmd := PTB_CmdState.cCMD_EJECTPAPER;
	CIf.Job.aCmdList[iIdx].strName := 'EJECTPAPER'; 
	CIf.Job.aCmdList[iIdx].bolAvailable := TRUE;
	iIdx := iIdx + 1;
	CIf.Job.aCmdList[iIdx].intCmd := PTB_CmdState.cCMD_STACKPAPER;
	CIf.Job.aCmdList[iIdx].strName := 'STACKPAPER'; 
	CIf.Job.aCmdList[iIdx].bolAvailable := TRUE;
ELSE
	// Error if the aCmdList Array is to small
END_IF

// set name of class/typ
CIf.Info.strType := 'FB_PTB';
CIf.Info.strFullName := 'Paper Transport Belt';

// set alarm class
SIf.Alm[E_ALM_PTB.TestAlarm].eAlmClass := Base_PLC.E_AlmClass.TSTOP;
SIf.Alm[E_ALM_PTB.TestAlarm].strText := 'Baum' ;


//*******************************************************************************
// initial values
//*******************************************************************************

// software configuration
CIf.SwCfg.bolExist := TRUE;
CIf.SwCfg.bolEnable := TRUE;
CIf.SwCfg.bolSimulation := FALSE;

// configuration
SIf.Cfg.rBeltParam.intBackwardDirection		:= E_TURN_DIRECTION.LEFT;
SIf.Cfg.rBeltParam.intForwardDirection		:= E_TURN_DIRECTION.RIGHT;
SIf.Cfg.bolVacuumPresent					:= TRUE;
SIf.Cfg.eMode								:= E_PTB_MODE.Endless;
SIf.Cfg.rBeltParam.reaRpmDistance_mm		:= 20.3;

// parameter
SIf.Par.intDirection				:= E_BELT_DIRECTION.FORWARD;
SIf.Par.rBeltParam.uinBeltSpeed		:= 412;
SIf.Par.udiDistanceToMove_mm		:= 0;
SIf.Par.udiTimeToMove_ms			:= 0;
SIf.Par.ePaperOrientation			:= E_PTB_PaperDirection.Portrait;
SIf.Par.uinPaperHight_mm			:= 460;
SIf.Par.uinPaperWidth_mm			:= 320;
SIf.Par.uinInputSignalDebounceTime_ms := 50;


fbEntrySensorDebounce.CtrlSIf^.Par.udiDebounceAbsentTime_ms := SIf.Par.uinInputSignalDebounceTime_ms;
fbEntrySensorDebounce.CtrlSIf^.Par.udiDebouncePresentTime_ms := SIf.Par.uinInputSignalDebounceTime_ms;
fbExitSensorDebounce.CtrlSIf^.Par.udiDebounceAbsentTime_ms := SIf.Par.uinInputSignalDebounceTime_ms;
fbExitSensorDebounce.CtrlSIf^.Par.udiDebouncePresentTime_ms := SIf.Par.uinInputSignalDebounceTime_ms;
END_METHOD

METHOD PROTECTED getCmdState : STRING

VAR_INPUT
	intCmdState: INT;
	bolState: BOOL;
END_VAR
getCmdState := SUPER^.getCmdState(intCmdState:=intCmdState,bolState:=bolState); // get global/base defined cmds/states

IF (getCmdState='') THEN // global not defined get local
	// get string cmd/state string information in runtime
	IF (bolState=FALSE) THEN
		CASE intCmdState OF
			PTB_CmdState.cCMD_EJECTPAPER: 
				getCmdState := 'EJECTPAPER';
			PTB_CmdState.cCMD_STACKPAPER: 
				getCmdState := 'STACKPAPER';
		END_CASE;
	ELSE
		// States's
		CASE intCmdState OF
			PTB_CmdState.cSTA_EJECTPAPER: 
				getCmdState := 'EJECTPAPER';
			PTB_CmdState.cSTA_EJECTPAPERbusy: 
				getCmdState := 'EJECTPAPERbusy';
			PTB_CmdState.cSTA_STACKPAPER: 
				getCmdState := 'STACKPAPER';
			PTB_CmdState.cSTA_STACKPAPERbusy: 
				getCmdState := 'STACKPAPERbusy';
			PTB_CmdState.cSUB_EMPTYstart: 
				getCmdState := 'EMPTYstart';
			PTB_CmdState.cSUB_EMPTYWAITPAPERbusy: 
				getCmdState := 'EMPTYWAITPAPERbusy';
			PTB_CmdState.cSUB_EMPTYWAITPAPERGONEbusy: 
				getCmdState := 'EMPTYWAITPAPERGONEbusy';
			PTB_CmdState.cSUB_PAPERDISTANCEbusy: 
				getCmdState := 'PAPERDISTANCEbusy';
			PTB_CmdState.cSUB_PAPERDISTANCEstart: 
				getCmdState := 'PAPERDISTANCEstart';
			PTB_CmdState.cSUB_STARTENTRYDRIVE: 
				getCmdState := 'STARTENTRYDRIVE';
			PTB_CmdState.cSUB_STARTENTRYDRIVEbusy: 
				getCmdState := 'STARTENTRYDRIVEbusy';
			PTB_CmdState.cSUB_STARTSTACKDELAY: 
				getCmdState := 'STARTSTACKDELAY';
			PTB_CmdState.cSUB_WAITPAPER: 
				getCmdState := 'WAITPAPER';
			PTB_CmdState.cSUB_PAPERDISTANCESTOPbusy:
				getCmdState := 'PAPERDISTANCESTOPbusy';
		END_CASE;
	END_IF
END_IF
END_METHOD

METHOD getCtrlSIf : POINTER TO T_Ctrl_SIf_PTB
getCtrlSIf := ADR(SIf);
END_METHOD

METHOD PROTECTED IoInBridge : BOOL
// digitale and analoge inputs read from hardware or forcing
IF SIf.Cfg.bolExitSensorDebounceEnable THEN
	fbExitSensorDebounce.In_bolPresent := THIS^.In_bolBeltExitSensor;
	fbExitSensorDebounce();
	SIf.In.bolBeltExitSensor.map := fbExitSensorDebounce.Out_bolPresent;
ELSE
	SIf.In.bolBeltExitSensor.map := THIS^.In_bolBeltExitSensor;
END_IF

IF SIf.Cfg.bolEntrySensorDebounceEnable THEN
	fbEntrySensorDebounce.In_bolPresent := THIS^.In_bolBeltExitSensor;
	fbEntrySensorDebounce();
	SIf.In.bolBeltExitSensor.map := fbEntrySensorDebounce.Out_bolPresent;
ELSE
	SIf.In.bolBeltEntrySensor.map := THIS^.In_bolBeltEntrySensor;
END_IF


// Insert also an edge detection
fbPaperEntryPEdge.CLK := SIf.In.bolBeltEntrySensor.map;
fbPaperEntryPEdge();
SIf.In.bolBeltEntrySensorPEdge.map := fbPaperEntryPEdge.Q;

fbPaperEntryNEdge.CLK := SIf.In.bolBeltEntrySensor.map;
fbPaperEntryNEdge();
SIf.In.bolBeltEntrySensorNEdge.map := fbPaperEntryNEdge.Q;

fbPaperExitPEdge.CLK := SIf.In.bolBeltExitSensor.map;
fbPaperExitPEdge();
SIf.In.bolBeltExitSensorPEdge.map := fbPaperExitPEdge.Q;

fbPaperExitNEdge.CLK := SIf.In.bolBeltExitSensor.map;
fbPaperExitNEdge();
SIf.In.bolBeltExitSensorNEdge.map := fbPaperExitNEdge.Q;

IF (CIf.SwCfg.bolSimulation = FALSE) THEN
	getInBol(CIf.Job.bolIoForce,ADR(SIf.In.bolBeltExitSensor));
	getInBol(CIf.Job.bolIoForce,ADR(SIf.In.bolBeltEntrySensor));
	getInBol(CIf.Job.bolIoForce,ADR(SIf.In.bolBeltEntrySensorPEdge));
	getInBol(CIf.Job.bolIoForce,ADR(SIf.In.bolBeltEntrySensorNEdge));
	getInBol(CIf.Job.bolIoForce,ADR(SIf.In.bolBeltExitSensorPEdge));
	getInBol(CIf.Job.bolIoForce,ADR(SIf.In.bolBeltExitSensorNEdge));
ELSE
;	//simulation of global IO
END_IF
END_METHOD

METHOD PROTECTED IoOutBridge : BOOL
VAR
	bolSwitchValvesOff: BOOL;
END_VAR
// digitale and analoge inputs read from hardware or forcing
IF (CIf.SwCfg.bolSimulation = FALSE) THEN
//	setOutBol(CIf.Job.bolIoForce ,ADR(SIf.Out.intActualPosition));
;
//	THIS^.Out_intActualPosition := SIf.Out.intActualPosition.map;
END_IF
END_METHOD

METHOD PROTECTED PaperPositionHandling : BOOL
VAR_INPUT
END_VAR
// Paper Tracking Service
// -----------------------------------------------------------------------------------
CASE me.StateMachine.intState OF
	BASE_PLC.cSTA_RUN:
		fbPositionService.In_uinBeltSpeed := sif.Cur.rBeltParam.uinBeltSpeed_mms;
ELSE
	fbPositionService.In_uinBeltSpeed := 0;
END_CASE

IF SIf.In.bolBeltEntrySensorPEdge.intern THEN
	udiIdCounter := udiIdCounter + 1;
	fbPositionService.Push(udiIdCounter);
END_IF

IF SIf.In.bolBeltEntrySensorNEdge.intern THEN
	fbPositionService.EnterComplete();
END_IF

IF SIf.In.bolBeltExitSensorPEdge.intern THEN
	fbPositionService.Pop();
END_IF

// Cyclic call
fbPositionService();
SIf.Cur.uinPaperOnBelt := fbPositionService.PaperOnBelt;
END_METHOD

PROPERTY PUBLIC PositionList : POINTER TO T_PTR_STRUCT
GET
END_GET
SET
END_SET
END_PROPERTY

METHOD PROTECTED SetPumpComand : BOOL
VAR_INPUT
	intComand		: INT;
END_VAR
SetPumpComand := TRUE;

IF SIf.Cfg.bolVacuumPresent THEN
	p_fbPump^.CtrlCIf^.Job.intACmd := intComand;
END_IF
END_METHOD

METHOD PROTECTED sta_EJECTPAPER : Bool
VAR
	iDifference 		: INT;
END_VAR
// state implemetation
//--------------------------------------------------------------------------------------
// Entry action
	IF (me.StateMachine.intState<>me.StateMachine.intStateLastCycle) THEN
		me.StateMachine.intStateLastCycle := me.StateMachine.intState;
	END_IF


//--------------------------------------------------------------------------------------
// Cyclic action
	IF (me.StateMachine.intState = me.StateMachine.intStateLastCycle) THEN
		CASE me.intCmd OF
			BASE_PLC.cCMD_RUN:
				me.StateMachine.intStateNext := BASE_PLC.cSTA_RUNBusy;
			BASE_PLC.cCMD_STOP:
				me.StateMachine.intStateNext := BASE_PLC.cSTA_STOPBusy;
			PTB_CmdState.cCMD_EJECTPAPER:
				me.StateMachine.intStateNext := PTB_CmdState.cSTA_EJECTPAPERbusy;
			PTB_CmdState.cCMD_STACKPAPER:
				me.StateMachine.intStateNext := PTB_CmdState.cSTA_STACKPAPERbusy;
		END_CASE
	END_IF

//--------------------------------------------------------------------------------------
// Exit action
	IF (me.StateMachine.intState<>me.StateMachine.intStateNext) THEN
		;
	END_IF
END_METHOD

METHOD PROTECTED sta_EJECTPAPERbusy : BOOL
VAR_INPUT
END_VAR
// state implemetation
//--------------------------------------------------------------------------------------
// Entry action
	IF (me.StateMachine.intState<>me.StateMachine.intStateLastCycle) THEN
		me.StateMachine.intStateLastCycle := me.StateMachine.intState;
		cmd_RUN(sif.Par.rBeltParam.uinBeltSpeed);
		me.SubStateMachine.intStateNext := PTB_CmdState.cSUB_EMPTYWAITPAPERbusy;
	END_IF


//--------------------------------------------------------------------------------------
// Cyclic action
	IF (me.StateMachine.intState=me.StateMachine.intStateLastCycle) THEN
		CASE me.SubStateMachine.intState OF
			PTB_CmdState.cSUB_EMPTYWAITPAPERbusy:
				IF SIf.In.bolBeltExitSensor.intern THEN
					me.SubStateMachine.intStateNext := PTB_CmdState.cSUB_EMPTYWAITPAPERGONEbusy;
				END_IF
			PTB_CmdState.cSUB_EMPTYWAITPAPERGONEbusy:
				IF NOT SIf.In.bolBeltExitSensor.intern THEN
					SIf.Cur.uinPaperOnBelt := 0;
					cmd_STOP();
					me.SubStateMachine.intStateNext := PTB_CmdState.cSUB_EMPTYWAITDRIVESTOPED;
				END_IF
			PTB_CmdState.cSUB_EMPTYWAITDRIVESTOPED:
				IF (p_fbMotor^.CtrlCIf^.Job.intState = BASE_PLC.cSTA_STOP) THEN
					IF SIf.Par.bolAutoStackAfterEject THEN
						CIf.Job.intACmd := BASE_PLC.cCMD_DONE;
						CIf.Job.intMCmd := BASE_PLC.cCMD_DONE;
						me.StateMachine.intStateNext := PTB_CmdState.cSTA_STACKPAPERbusy;	
					ELSE	
						me.StateMachine.intStateNext := PTB_CmdState.cSTA_EJECTPAPER;	
					END_IF
				END_IF
		END_CASE
	END_IF


//--------------------------------------------------------------------------------------
// Exit action
	IF (me.StateMachine.intState<>me.StateMachine.intStateNext) THEN
		me.SubStateMachine.intState := BASE_PLC.cSTA_INITIALIZED;
	END_IF
END_METHOD

METHOD PROTECTED sta_ERROR : BOOL
// state implemetation
//--------------------------------------------------------------------------------------
// Entry action
	IF (me.StateMachine.intState<>me.StateMachine.intStateLastCycle) THEN
		me.StateMachine.intStateHistory := me.StateMachine.intStateLastCycle; // -> possibillity to go back to state before error
		me.StateMachine.intStateLastCycle := me.StateMachine.intState;
		pMotorCIf^.Job.intACmd := BASE_PLC.cCMD_OFF;		
	END_IF


//--------------------------------------------------------------------------------------
// Cyclic action
	IF (me.StateMachine.intState=me.StateMachine.intStateLastCycle) THEN
		
		;
		
		
		// State Change Condition
		IF (CIf.Job.bolAlmReset = TRUE) THEN
			me.StateMachine.intStateNext := cSTA_ERRORQuit;
		END_IF
	END_IF




//--------------------------------------------------------------------------------------
// Exit action
	IF (me.StateMachine.intState<>me.StateMachine.intStateNext) THEN
		;
	END_IF
END_METHOD

METHOD PROTECTED sta_ERRORQuit : BOOL
// state implemetation
//--------------------------------------------------------------------------------------
// Entry action
	IF (me.StateMachine.intState<>me.StateMachine.intStateLastCycle) THEN
		me.StateMachine.intStateLastCycle := me.StateMachine.intState;
		
	END_IF


//--------------------------------------------------------------------------------------
// Cyclic action
	IF (me.StateMachine.intState=me.StateMachine.intStateLastCycle) THEN
		
		;
		// evtl. wait time if reset of device is necessary and then decide to go to states or ERROR state
		IF (CIf.Job.bolAlmReset = TRUE) THEN
			CIf.Job.eMe_ActivAlmClass := E_AlmClass.NONE; // reset feedback channel for parent
			CIf.Job.bolAlmReset := FALSE;
		END_IF
		
		// State Change Condition
		IF (CIf.Job.bolAlmReset = FALSE) THEN
			IF (me.StateMachine.intStateHistory<=cSTA_PON) THEN
				me.StateMachine.intStateNext := cSTA_PONBusy;
			ELSIF(me.intCmd=cCMD_OFF) THEN
				me.StateMachine.intStateNext := cSTA_OFFBusy;
			ELSIF(me.intCmd=BASE_PLC.cCMD_RUN) THEN
				me.StateMachine.intStateNext := BASE_PLC.cSTA_RUNBusy;
			END_IF
		END_IF
	END_IF




//--------------------------------------------------------------------------------------
// Exit action
	IF (me.StateMachine.intState<>me.StateMachine.intStateNext) THEN
		;
	END_IF
END_METHOD

METHOD PROTECTED sta_OFF : BOOL
VAR_INPUT
END_VAR
// state implemetation
//--------------------------------------------------------------------------------------
// Entry action
	IF (me.StateMachine.intState<>me.StateMachine.intStateLastCycle) THEN
		me.StateMachine.intStateLastCycle := me.StateMachine.intState;
	END_IF


//--------------------------------------------------------------------------------------
// Cyclic action
	IF (me.StateMachine.intState=me.StateMachine.intStateLastCycle) THEN
		CASE me.intCmd OF
			BASE_PLC.cCMD_RUN:
				me.StateMachine.intStateNext := BASE_PLC.cSTA_RUNBusy;
			BASE_PLC.cCMD_STOP:
				me.StateMachine.intStateNext := BASE_PLC.cSTA_STOPBusy;
			PTB_CmdState.cCMD_EJECTPAPER:
				me.StateMachine.intStateNext := PTB_CmdState.cSTA_EJECTPAPERbusy;
			PTB_CmdState.cCMD_STACKPAPER:
				me.StateMachine.intStateNext := PTB_CmdState.cSTA_STACKPAPERbusy;
		END_CASE
	END_IF


//--------------------------------------------------------------------------------------
// Exit action
	IF (me.StateMachine.intState<>me.StateMachine.intStateNext) THEN
		;
	END_IF
END_METHOD

METHOD PROTECTED sta_OFFBusy : BOOL
VAR_INPUT
END_VAR
// state implemetation
//--------------------------------------------------------------------------------------
// Entry action
	IF (me.StateMachine.intState<>me.StateMachine.intStateLastCycle) THEN
		me.StateMachine.intStateLastCycle := me.StateMachine.intState;
		cmd_OFF();
	END_IF


//--------------------------------------------------------------------------------------
// Cyclic action
	IF (me.StateMachine.intState=me.StateMachine.intStateLastCycle) THEN

		// Set commandos not only in entry action because of possible errors or manual/auto changes
		cmd_OFF();

		IF p_fbMotor^.CtrlCIf^.Job.intState = BASE_PLC.cSTA_OFF 
		  AND CheckPumpState(BASE_PLC.cSTA_OFF) THEN
			me.StateMachine.intStateNext := BASE_PLC.cSTA_OFF;
		END_IF
	END_IF


//--------------------------------------------------------------------------------------
// Exit action
	IF (me.StateMachine.intState<>me.StateMachine.intStateNext) THEN
		;
	END_IF
END_METHOD

METHOD PROTECTED sta_PON : BOOL
VAR_INPUT
END_VAR
// state implemetation
//--------------------------------------------------------------------------------------
// Entry action
	IF (me.StateMachine.intState<>me.StateMachine.intStateLastCycle) THEN
		me.StateMachine.intStateLastCycle := me.StateMachine.intState;
		
	END_IF


//--------------------------------------------------------------------------------------
// Cyclic action
	IF (me.StateMachine.intState=me.StateMachine.intStateLastCycle) THEN
		;
	END_IF




//--------------------------------------------------------------------------------------
// Exit action
	IF (me.StateMachine.intState<>me.StateMachine.intStateNext) THEN
		;
	END_IF
END_METHOD

METHOD PROTECTED sta_RUN : Bool
VAR
	iDifference 		: INT;
END_VAR
// state implemetation
//--------------------------------------------------------------------------------------
// Entry action
	IF (me.StateMachine.intState<>me.StateMachine.intStateLastCycle) THEN
		me.StateMachine.intStateLastCycle := me.StateMachine.intState;
	END_IF


//--------------------------------------------------------------------------------------
// Cyclic action
	IF (me.StateMachine.intState = me.StateMachine.intStateLastCycle) THEN
		// The direction changed
		IF (SIf.Par.intDirection <> SIf.Cur.eActualDirection) THEN
			me.StateMachine.intStateNext := BASE_PLC.cSTA_RUNBusy;
		END_IF
		
		// The speed changed
		IF (SIf.Par.rBeltParam.uinBeltSpeed <> SIf.Cur.rBeltParam.uinBeltSpeed_mms) THEN
			me.StateMachine.intStateNext := BASE_PLC.cSTA_RUNBusy;
		END_IF
		
		IF  me.intCmd = BASE_PLC.cCMD_STOP THEN
			me.StateMachine.intStateNext := BASE_PLC.cSTA_STOPBusy;
		END_IF

		CASE SIf.Cfg.eMode OF
			E_PTB_MODE.ToDistance, 
			E_PTB_MODE.ToTime :
				IF me.StateMachine.udiTimeInState_ms > SIf.Cur.udiTimeToMove_ms THEN
					me.StateMachine.intStateNext := BASE_PLC.cSTA_STOPBusy;
				END_IF
			E_PTB_MODE.ToSensor:
				IF (SIf.In.bolBeltExitSensorPEdge.intern) THEN
					me.StateMachine.intStateNext := BASE_PLC.cSTA_STOPBusy;
				END_IF
		END_CASE
	END_IF


//--------------------------------------------------------------------------------------
// Exit action
	IF (me.StateMachine.intState<>me.StateMachine.intStateNext) THEN
		;
	END_IF
END_METHOD

METHOD PROTECTED sta_RUNBusy : BOOL
VAR_INPUT
END_VAR
// state implemetation
//--------------------------------------------------------------------------------------
// Entry action
	IF (me.StateMachine.intState<>me.StateMachine.intStateLastCycle) THEN
		me.StateMachine.intStateLastCycle := me.StateMachine.intState;
		
		CASE SIf.Cfg.eMode OF
			E_PTB_MODE.Endless,
			E_PTB_MODE.ToDistance,
			E_PTB_MODE.ToTime:
				cmd_RUN(sif.Par.rBeltParam.uinBeltSpeed);
			E_PTB_MODE.ToSensor:
				IF SIf.In.bolBeltExitSensorPEdge.intern THEN
					me.StateMachine.intStateNext := BASE_PLC.cSTA_STOPBusy;
				ELSE
					cmd_RUN(sif.Par.rBeltParam.uinBeltSpeed);
				END_IF
		END_CASE
	END_IF


//--------------------------------------------------------------------------------------
// Cyclic action
	IF (me.StateMachine.intState=me.StateMachine.intStateLastCycle) THEN
		IF (p_fbMotor^.CtrlCIf^.Job.intState = BASE_PLC.cSTA_RUN) 
		  AND (p_fbMotor^.CtrlSIf^.Cur.eDirection = arMotorDirection[SIf.Par.intDirection]) 
		  AND CheckPumpState(BASE_PLC.cSTA_RUN) THEN
			me.StateMachine.intStateNext := BASE_PLC.cSTA_RUN;
		END_IF

		IF me.intCmd = BASE_PLC.cCMD_STOP THEN
			me.StateMachine.intStateNext := BASE_PLC.cSTA_STOPBusy;
		END_IF
	END_IF


//--------------------------------------------------------------------------------------
// Exit action
	IF (me.StateMachine.intState<>me.StateMachine.intStateNext) THEN
		;
	END_IF
END_METHOD

METHOD PROTECTED sta_STACKPAPER : Bool
VAR
END_VAR
// state implemetation
//--------------------------------------------------------------------------------------
// Entry action
	IF (me.StateMachine.intState<>me.StateMachine.intStateLastCycle) THEN
		me.StateMachine.intStateLastCycle := me.StateMachine.intState;
	END_IF


//--------------------------------------------------------------------------------------
// Cyclic action
	IF (me.StateMachine.intState = me.StateMachine.intStateLastCycle) THEN
		CASE me.intCmd OF
			BASE_PLC.cCMD_RUN:
				me.StateMachine.intStateNext := BASE_PLC.cSTA_RUNBusy;
			BASE_PLC.cCMD_STOP:
				me.StateMachine.intStateNext := BASE_PLC.cSTA_STOPBusy;
			PTB_CmdState.cCMD_EJECTPAPER:
				me.StateMachine.intStateNext := PTB_CmdState.cSTA_EJECTPAPERbusy;
			PTB_CmdState.cCMD_STACKPAPER:
				me.StateMachine.intStateNext := PTB_CmdState.cSTA_STACKPAPERbusy;
		END_CASE
	END_IF


//--------------------------------------------------------------------------------------
// Exit action
	IF (me.StateMachine.intState<>me.StateMachine.intStateNext) THEN
		;
	END_IF
END_METHOD

METHOD PROTECTED sta_STACKPAPERbusy : BOOL
VAR_INPUT
END_VAR
// state implemetation
//--------------------------------------------------------------------------------------
// Entry action
	IF (me.StateMachine.intState<>me.StateMachine.intStateLastCycle) THEN
		me.StateMachine.intStateLastCycle := me.StateMachine.intState;

		me.SubStateMachine.intStateNext := PTB_CmdState.cSUB_WAITPAPER;
	END_IF


//--------------------------------------------------------------------------------------
// Cyclic action
	IF (me.StateMachine.intState=me.StateMachine.intStateLastCycle) THEN
		CASE me.SubStateMachine.intState OF
			PTB_CmdState.cSUB_WAITPAPER:
				IF SIf.In.bolBeltEntrySensor.intern THEN
					me.SubStateMachine.intStateNext := PTB_CmdState.cSUB_WAITPAPERGONE;
				ELSE
					CASE me.intCmd OF
						BASE_PLC.cCMD_RUN:
							me.StateMachine.intStateNext := BASE_PLC.cSTA_RUNBusy;
						BASE_PLC.cCMD_STOP:
							me.StateMachine.intStateNext := BASE_PLC.cSTA_STOPBusy;
						PTB_CmdState.cCMD_EJECTPAPER:
							me.StateMachine.intStateNext := PTB_CmdState.cSTA_EJECTPAPERbusy;
					END_CASE
				END_IF
			PTB_CmdState.cSUB_WAITPAPERGONE:
				IF NOT SIf.In.bolBeltEntrySensor.intern THEN
					SIf.Cur.uinPaperOnBelt := SIf.Cur.uinPaperOnBelt + 1;
					me.SubStateMachine.intStateNext := PTB_CmdState.cSUB_STARTSTACKDELAY;
				END_IF
			PTB_CmdState.cSUB_STARTSTACKDELAY:
				IF me.SubStateMachine.udiTimeInState_ms > SIf.Par.udiStackDelayTime_ms THEN
					IF SIf.Cur.uinPaperOnBelt >= SIf.Par.uinPaperStackHight THEN
						me.StateMachine.intStateNext := PTB_CmdState.cSTA_EJECTPAPERbusy;
					ELSE
						me.SubStateMachine.intStateNext := PTB_CmdState.cSUB_PAPERDISTANCEstart;
					END_IF
				END_IF
			PTB_CmdState.cSUB_PAPERDISTANCEstart:
				cmd_RUN(sif.Par.rBeltParam.uinStackSpeed);
				me.SubStateMachine.intStateNext := PTB_CmdState.cSUB_PAPERDISTANCEbusy;
			PTB_CmdState.cSUB_PAPERDISTANCEbusy:
				IF me.SubStateMachine.udiTimeInState_ms > SIf.Cur.udiTimeToMove_ms THEN
					cmd_STOP();
					me.SubStateMachine.intStateNext := PTB_CmdState.cSUB_PAPERDISTANCESTOPbusy;
				END_IF
			PTB_CmdState.cSUB_PAPERDISTANCESTOPbusy:
				IF p_fbMotor^.CtrlCIf^.Job.intState = BASE_PLC.cSTA_STOP THEN
					IF SIf.Par.bolAutoEjectAfterStack THEN
						me.StateMachine.intStateNext := PTB_CmdState.cSTA_EJECTPAPERbusy;
					ELSE
						me.StateMachine.intStateNext := PTB_CmdState.cSTA_STACKPAPER;
					END_IF
				END_IF
		END_CASE
	END_IF


//--------------------------------------------------------------------------------------
// Exit action
	IF (me.StateMachine.intState<>me.StateMachine.intStateNext) THEN
		CIf.Job.intACmd := BASE_PLC.cCMD_DONE;
		CIf.Job.intMCmd := BASE_PLC.cCMD_DONE;
		me.SubStateMachine.intState := BASE_PLC.cSTA_INITIALIZED;
	END_IF
END_METHOD

METHOD PROTECTED sta_STOP : BOOL
VAR_INPUT
END_VAR
// state implemetation
//--------------------------------------------------------------------------------------
// Entry action
	IF (me.StateMachine.intState<>me.StateMachine.intStateLastCycle) THEN
		me.StateMachine.intStateLastCycle := me.StateMachine.intState;
	END_IF


//--------------------------------------------------------------------------------------
// Cyclic action
	IF (me.StateMachine.intState=me.StateMachine.intStateLastCycle) THEN
		CASE me.intCmd OF
			BASE_PLC.cCMD_RUN:
				me.StateMachine.intStateNext := BASE_PLC.cSTA_RUNBusy;
			BASE_PLC.cCMD_STOP:
				me.StateMachine.intStateNext := BASE_PLC.cSTA_STOPBusy;
			PTB_CmdState.cCMD_EJECTPAPER:
				me.StateMachine.intStateNext := PTB_CmdState.cSTA_EJECTPAPERbusy;
			PTB_CmdState.cCMD_STACKPAPER:
				me.StateMachine.intStateNext := PTB_CmdState.cSTA_STACKPAPERbusy;
		END_CASE

		IF    (SIf.Cfg.eMode = E_PTB_MODE.ToSensor) 
		  AND (SIf.In.bolBeltExitSensorNEdge.intern) THEN
			me.StateMachine.intStateNext := BASE_PLC.cSTA_RUNBusy;
		END_IF
	END_IF


//--------------------------------------------------------------------------------------
// Exit action
	IF (me.StateMachine.intState<>me.StateMachine.intStateNext) THEN
		;
	END_IF
END_METHOD

METHOD PROTECTED sta_STOPBusy : BOOL
VAR_INPUT
END_VAR
// state implemetation
//--------------------------------------------------------------------------------------
// Entry action
	IF (me.StateMachine.intState<>me.StateMachine.intStateLastCycle) THEN
		me.StateMachine.intStateLastCycle := me.StateMachine.intState;
		cmd_STOP();
	END_IF


//--------------------------------------------------------------------------------------
// Cyclic action
	IF (me.StateMachine.intState=me.StateMachine.intStateLastCycle) THEN
		IF p_fbMotor^.CtrlCIf^.Job.intState = BASE_PLC.cSTA_STOP  THEN
			me.StateMachine.intStateNext := BASE_PLC.cSTA_STOP;
		END_IF
	END_IF


//--------------------------------------------------------------------------------------
// Exit action
	IF (me.StateMachine.intState<>me.StateMachine.intStateNext) THEN
		;
	END_IF
END_METHOD

METHOD PROTECTED StateMachine : BOOL
SUPER^.StateMachine();

// main statemachine of base controller
CASE me.StateMachine.intState OF
    BASE_PLC.cSTA_RUN: 
        THIS^.sta_RUN();
    BASE_PLC.cSTA_RUNBusy: 
        THIS^.sta_RUNBusy();
    BASE_PLC.cSTA_STOP: 
        THIS^.sta_STOP();
    BASE_PLC.cSTA_STOPBusy: 
        THIS^.sta_STOPBusy();
	PTB_CmdState.cSTA_EJECTPAPERbusy:
		THIS^.sta_EJECTPAPERbusy();
	PTB_CmdState.cSTA_EJECTPAPER:
		THIS^.sta_EJECTPAPER();
	PTB_CmdState.cSTA_STACKPAPER:
		THIS^.sta_STACKPAPER();
	PTB_CmdState.cSTA_STACKPAPERbusy:
		THIS^.sta_STACKPAPERbusy();
END_CASE;
END_METHOD

PROPERTY PUBLIC VacuumPump :  POINTER TO FB_VPC
GET
VacuumPump := p_fbPump;
END_GET
SET
p_fbPump := VacuumPump;
END_SET
END_PROPERTY

END_FUNCTION_BLOCK

// POUs/Controller/Lvl2/PBC [Paper Buffer Controller]/helper/cycle_Pbc
FUNCTION cycle_Pbc : BOOL
VAR_INPUT
	pPbc: POINTER TO T_PBC;
END_VAR

pPbc^.ctrl.fbPbc_PtbDeStacker_Umc.In_bolEmoOk 				:= pPbc^.io.In_bolPtbDeStacker_Umc_EmoOk;
pPbc^.ctrl.fbPbc_PtbDeStacker_Umc.In_uinStatus 				:= pPbc^.io.In_uinPtbDeStacker_Umc_Status;
pPbc^.ctrl.fbPbc_PtbDeStacker_Umc.In_intMotorActualSpeed 	:= pPbc^.io.In_uinPtbDeStacker_Umc_ActualSpeed;
pPbc^.ctrl.fbPbc_PtbDeStacker_Umc.In_uinMotorSetSpeed 		:= pPbc^.io.In_uinPtbDeStacker_Umc_SetSpeed;
pPbc^.ctrl.fbPbc_PtbDeStacker_Umc.In_uinECATState 			:= pPbc^.io.In_uinPtbDeStacker_Umc_ECatState;
pPbc^.ctrl.fbPbc_PtbDeStacker_Umc.In_strNetId 				:= pPbc^.io.In_strPtbDeStacker_Umc_ECatNetId;
pPbc^.ctrl.fbPbc_PtbDeStacker_Umc.In_uintPort 				:= pPbc^.io.In_uinPtbDeStacker_Umc_ECatPort;
pPbc^.ctrl.fbPbc_PtbDeStacker_Umc();
pPbc^.io.Out_uinPtbDeStacker_Umc_SetSpeed	 				:= pPbc^.ctrl.fbPbc_PtbDeStacker_Umc.Out_uinSpeedSetpoint;
pPbc^.io.Out_uinPtbDeStacker_Umc_Control 					:= pPbc^.ctrl.fbPbc_PtbDeStacker_Umc.Out_uinControl;

pPbc^.ctrl.fbPbc_PtbDeStacker();

pPbc^.ctrl.fbPbc_PtbBelt_Umc.In_bolEmoOk 					:= pPbc^.io.In_bolPtbBelt_Umc_EmoOk;
pPbc^.ctrl.fbPbc_PtbBelt_Umc.In_uinStatus 					:= pPbc^.io.In_uinPtbBelt_Umc_Status;
pPbc^.ctrl.fbPbc_PtbBelt_Umc.In_intMotorActualSpeed 		:= pPbc^.io.In_uinPtbBelt_Umc_ActualSpeed;
pPbc^.ctrl.fbPbc_PtbBelt_Umc.In_uinMotorSetSpeed 			:= pPbc^.io.In_uinPtbBelt_Umc_SetSpeed;
pPbc^.ctrl.fbPbc_PtbBelt_Umc.In_uinECATState 				:= pPbc^.io.In_uinPtbBelt_Umc_ECatState;
pPbc^.ctrl.fbPbc_PtbBelt_Umc.In_strNetId 					:= pPbc^.io.In_strPtbBelt_Umc_ECatNetId;
pPbc^.ctrl.fbPbc_PtbBelt_Umc.In_uintPort 					:= pPbc^.io.In_uinPtbBelt_Umc_ECatPort;
pPbc^.ctrl.fbPbc_PtbBelt_Umc();
pPbc^.io.Out_uinPtbBelt_Umc_SetSpeed 						:= pPbc^.ctrl.fbPbc_PtbBelt_Umc.Out_uinSpeedSetpoint;
pPbc^.io.Out_uinPtbBelt_Umc_Control 						:= pPbc^.ctrl.fbPbc_PtbBelt_Umc.Out_uinControl;

pPbc^.ctrl.fbPbc_PtbBelt_Vpc.In_bolPumpOk 					:= pPbc^.io.In_bolPtbBelt_Vpc_PumpOk;
pPbc^.ctrl.fbPbc_PtbBelt_Vpc.In_bolVacuumOk 				:= pPbc^.io.In_bolPtbBelt_Vpc_VacuumSensor;
pPbc^.ctrl.fbPbc_PtbBelt_Vpc();
pPbc^.io.Out_bolPtbBelt_Vpc_PumpOn 							:= pPbc^.ctrl.fbPbc_PtbBelt_Vpc.Out_bolVaccumPumpOn;

pPbc^.ctrl.fbPbc_PtbBelt();

pPbc^.ctrl.fbPbc.In_bolCapacityReached 						:= pPbc^.io.In_bolInputSensor;
pPbc^.ctrl.fbPbc.In_bolPaperAvailableEntry 					:= pPbc^.io.In_bolCapacitySensor;
pPbc^.ctrl.fbPbc.In_bolPaperAvailableExit 					:= pPbc^.io.In_bolOutputSensor;
pPbc^.ctrl.fbPbc.In_bolDoublePaperDetection 				:= pPbc^.io.In_bolDoublePaperSensor;
pPbc^.ctrl.fbPbc.In_bolTurnTableMiddleSensor 				:= pPbc^.io.In_bolPts_PaperSensor;
pPbc^.ctrl.fbPbc.In_bolAirPressorOk 						:= pPbc^.io.In_bolAirPressureOk;
pPbc^.ctrl.fbPbc();
pPbc^.io.Out_bolAirPressureOn 								:= pPbc^.ctrl.fbPbc.Out_bolAirOn;

END_FUNCTION

// POUs/Controller/Lvl2/PBC [Paper Buffer Controller]/helper/init_Pbc
FUNCTION init_Pbc : BOOL
VAR_INPUT
	pPbc			: POINTER TO T_PBC;
	/// instance array of all controller instances
	pCtrlInst		: POINTER TO fb_CtrlBase;
	/// common interface array of all controllers (main use for PLC)
	pCtrlCIf		: POINTER TO T_Ctrl_CIf;
END_VAR

pPbc^.ctrl.fbPbc_PtbDeStacker_Umc.iniAllCtrlArrays(pCtrlInst,pCtrlCIf,pPbc^.id.Pbc_PtbDeStacker_Umc); // init and entry fb_instance in global fb pointer array
pPbc^.ctrl.fbPbc_PtbDeStacker.iniAllCtrlArrays(pCtrlInst,pCtrlCIf,pPbc^.id.Pbc_PtbDeStacker); // init and entry fb_instance in global fb pointer array
pPbc^.ctrl.fbPbc_PtbDeStacker.Drive := ADR(pPbc^.ctrl.fbPbc_PtbDeStacker_Umc);

pPbc^.ctrl.fbPbc_PtbBelt_Umc.iniAllCtrlArrays(pCtrlInst,pCtrlCIf,pPbc^.id.Pbc_PtbBelt_Umc); // init and entry fb_instance in global fb pointer array
pPbc^.ctrl.fbPbc_PtbBelt_Vpc.iniAllCtrlArrays(pCtrlInst,pCtrlCIf,pPbc^.id.Pbc_PtbBelt_Vpc); // init and entry fb_instance in global fb pointer array
pPbc^.ctrl.fbPbc_PtbBelt.iniAllCtrlArrays(pCtrlInst,pCtrlCIf,pPbc^.id.Pbc_PtbBelt); // init and entry fb_instance in global fb pointer array
pPbc^.ctrl.fbPbc_PtbBelt.Drive := ADR(pPbc^.ctrl.fbPbc_PtbBelt_Umc);
pPbc^.ctrl.fbPbc_PtbBelt.VacuumPump := ADR(pPbc^.ctrl.fbPbc_PtbBelt_Vpc);

pPbc^.ctrl.fbPbc.iniAllCtrlArrays(pCtrlInst,pCtrlCIf,pPbc^.id.Pbc); 		 // init and entry fb_instance in global fb pointer array
pPbc^.ctrl.fbPbc.DeStacker := ADR(pPbc^.ctrl.fbPbc_PtbDeStacker);
pPbc^.ctrl.fbPbc.Belt := ADR(pPbc^.ctrl.fbPbc_PtbBelt);

END_FUNCTION

// POUs/Controller/Lvl2/PBC [Paper Buffer Controller]/FB_PBC
FUNCTION_BLOCK FB_PBC EXTENDS FB_CtrlBase
VAR_INPUT
	In_bolPaperAvailableExit: BOOL;
	In_bolPaperAvailableEntry: BOOL;
	In_bolCapacityReached: BOOL;
	In_bolDoublePaperDetection: BOOL;
	In_bolTurnTableMiddleSensor: BOOL;
	In_bolAirPressorOk: BOOL;
END_VAR
VAR_OUTPUT
	Out_bolAirOn: BOOL;
END_VAR
VAR
	/// Specific interface struct for public access
	/// -------------------------------------------------------
	SIf: T_Ctrl_SIf_PBC;
	///Sub Controller Pointer
	/// -------------------------------------------------------
	p_fbDeStacker: POINTER TO FB_PTB;
	pDeStackerCIf: POINTER TO BASE_PLC.T_Ctrl_CIf;
	p_fbBelt: POINTER TO FB_PTB;
	pBeltCIf: POINTER TO BASE_PLC.T_Ctrl_CIf;
	/// Other localy used variables
	/// -------------------------------------------------------
	m_uinPaperHight_mm: UINT := 460;
	m_uinPaperWidth_mm: UINT := 320;
	m_intRetry: INT := 0;
END_VAR
VAR CONSTANT
	cPAPERPOSITION_TOLERANCE_mm: UINT := 200;
END_VAR

(*__________________________________________________________________________________________________
¦	
¦	Vistaprint Schweiz GmbH
¦	CH - 8401 Winterthur
¦
¦	www.vistaprint.ch - info@vistaprint.ch
¦___________________________________________________________________________________________________

Function desription:
Destacker/Buffer implementation. 


History:
Version		Date			Author		Comment
---------------------------------------------------------------------------------------------------
0.00.1		09.07.2013		PC			Start history
___________________________________________________________________________________________________*)


SUPER^();

{attribute 'object_name' := 'Always'}
METHOD PROTECTED Always : BOOL
VAR
	pItem: POINTER TO T_IdBase_DCH;
	bResult: BOOL;
END_VAR
SUPER^.Always();

// ----------------------------------------------------------------------------------
// cyclic actions outside of statemachine
IF (me.StateMachine.intState<>cSTA_SINGLE_ANSWER) THEN
	;
END_IF

// ----------------------------------------------------------------------------------
// Conditions Always
IF (((me.Alarm.eActivAlmClass=E_AlmClass.EOFF) OR (me.Alarm.eActivAlmClass=E_AlmClass.OFF) OR (me.intCmd=cCMD_OFF) OR (me.intCmd=BASE_PLC.cCMD_EOFF))
		 AND (me.StateMachine.intState<>cSTA_ERROR) AND (me.StateMachine.intState<>cSTA_ERRORQuit) AND
		(me.StateMachine.intState<>cSTA_OFF) AND (me.StateMachine.intState<>cSTA_OFFBusy)) THEN
	// alarm evt EOFF, OFF or cmd off
	me.StateMachine.intStateNext := cSTA_OFFBusy;
END_IF
END_METHOD

PROPERTY Belt : POINTER TO FB_PTB
GET
Belt := p_fbBelt;
END_GET
SET
p_fbBelt := Belt;
END_SET
END_PROPERTY

{attribute 'object_name' := 'CountPaper'}
METHOD PROTECTED CountPaper : UINT
END_METHOD

{attribute 'object_name' := 'CtrlInit'}
METHOD CtrlInit : BOOL
VAR
	pBccSIf: POINTER TO T_Ctrl_SIf_BCC;
END_VAR
SUPER^.CtrlInit();

pDeStackerCIf 	:= AddChild(p_fbDeStacker^);
pBeltCIf 		:= AddChild(p_fbBelt^);
END_METHOD

PROPERTY CtrlSIf : POINTER TO T_Ctrl_SIf_PBC
GET
CtrlSIf := ADR(SIf);
END_GET
SET
END_SET
END_PROPERTY

PROPERTY DeStacker : POINTER TO FB_PTB
GET
DeStacker := p_fbDeStacker;
END_GET
SET
p_fbDeStacker := DeStacker;
END_SET
END_PROPERTY

{attribute 'object_name' := 'FB_init'}
METHOD FB_init : BOOL
VAR_INPUT
	/// if TRUE, the retain variables are initialized (warm start / cold start)
	bInitRetains: BOOL;
	/// if TRUE, the instance afterwards gets moved into the copy code (online change)
	bInCopyCode: BOOL;
END_VAR
VAR
	iIdx: UINT;
	iLength: UINT;
END_VAR
//------------------------------------------------------------------------------------------------------------------------
// to manually change in new FUB implementation!!!
// define valid commands for this controller
iLength := SIZEOF(CIf.Job.aCmdList)/SIZEOF(CIf.Job.aCmdList[0]);
iIdx := 0;

WHILE (iIdx < iLength) AND (CIf.Job.aCmdList[iIdx].intCmd <> cCMD_INITIALIZED) DO
	iIdx := iIdx + 1; 
END_WHILE

IF (iIdx < iLength) THEN
// Add configuration of own comands	
	CIf.Job.aCmdList[iIdx].intCmd := BASE_PLC.cCMD_RUN;
	CIf.Job.aCmdList[iIdx].strName := 'RUN'; 
	CIf.Job.aCmdList[iIdx].bolAvailable := TRUE;
	iIdx := iIdx + 1;
	CIf.Job.aCmdList[iIdx].intCmd := BASE_PLC.cCMD_STOP;
	CIf.Job.aCmdList[iIdx].strName := 'STOP'; 
	CIf.Job.aCmdList[iIdx].bolAvailable := TRUE;
	iIdx := iIdx + 1;
	CIf.Job.aCmdList[iIdx].intCmd := PBC_CmdState.cCMD_SINGLE;
	CIf.Job.aCmdList[iIdx].strName := 'SINGLE'; 
	CIf.Job.aCmdList[iIdx].bolAvailable := TRUE;
	iIdx := iIdx + 1;
	CIf.Job.aCmdList[iIdx].intCmd := PBC_CmdState.cCMD_STANDBY;
	CIf.Job.aCmdList[iIdx].strName := 'STANDBY'; 
	CIf.Job.aCmdList[iIdx].bolAvailable := TRUE;
ELSE
	// Error if the aCmdList Array is to small
END_IF

// set name of class/typ
CIf.Info.strType := 'FB_PBC';
CIf.Info.strFullName := 'Paper Buffer Controller';

// set alarm class
SIf.Alm[E_ALM_PBC.BufferEmpty].eAlmClass := Base_PLC.E_AlmClass.WARNING;
SIf.Alm[E_ALM_PBC.BufferEmpty].strText := 'Buffer is Empty'; 
SIf.Alm[E_ALM_PBC.BufferFull].eAlmClass := E_AlmClass.TSTOP;
SIf.Alm[E_ALM_PBC.BufferFull].strText := 'Buffer reached capacity limit';
SIf.Alm[E_ALM_PBC.PaperTransport].eAlmClass := E_AlmClass.TSTOP;
SIf.Alm[E_ALM_PBC.PaperTransport].strText := 'Possible Paper Jam';
SIf.Alm[E_ALM_PBC.DoublePaper].eAlmClass := E_AlmClass.TSTOP;
SIf.Alm[E_ALM_PBC.DoublePaper].strText := 'Double paper detected';
SIf.Alm[E_ALM_PBC.DataChannelBufferFull].eAlmClass := E_AlmClass.WARNING;
SIf.Alm[E_ALM_PBC.DataChannelBufferFull].strText := 'Data Channel buffer is full';
SIf.Alm[E_ALM_PBC.DataChannelSend].eAlmClass := E_AlmClass.WARNING;
SIf.Alm[E_ALM_PBC.DataChannelSend].strText := 'Data Channel item could not be sent';
SIf.Alm[E_ALM_PBC.PaperInject].eAlmClass := E_AlmClass.TSTOP;
SIf.Alm[E_ALM_PBC.PaperInject].strText := 'Paper is not transported to the front';
SIf.Alm[E_ALM_PBC.PaperInjectRetry].eAlmClass := E_AlmClass.WARNING;
SIf.Alm[E_ALM_PBC.PaperInjectRetry].strText := 'Paper transport retry';

//*******************************************************************************
// initial values
//*******************************************************************************

// software configuration
CIf.SwCfg.bolExist := TRUE;
CIf.SwCfg.bolEnable := TRUE;
CIf.SwCfg.bolSimulation := FALSE;

// Configuration
SIf.Cfg.bolUseTurnTableSensorForEject := TRUE;
SIf.Cfg.bolEnableDataChannel		  := FALSE;
SIf.Cfg.bolGranulatAirPressureUnitAvailable := FALSE;

// parameter
SIf.Par.bolAutomaticMode := FALSE;
SIf.Par.udiPaperTransportTime := 3000;
SIf.Par.udiSheetToEject := 1;
SIf.Par.udiSheetToSheetTime := 5000;
SIf.Par.udiPaperInjectRetryPauseTime_ms := 400;
SIf.Par.udiPaperInjectRetries := 3;
SIf.Par.udiDoublePaperDebounceTime_ms := 500;
SIf.Par.bolEnableDoublePaperDetection := FALSE;
SIf.Par.udiSimPaperTransportTime := SIf.Par.udiPaperTransportTime / 2;
SIf.Par.udiSimPaperToPaperTransportTime := SIf.Par.udiPaperTransportTime / 20;
END_METHOD

{attribute 'object_name' := 'getCmdState'}
METHOD PROTECTED getCmdState : STRING
VAR_INPUT
	intCmdState: INT;
	bolState: BOOL;
END_VAR
getCmdState := SUPER^.getCmdState(intCmdState:=intCmdState,bolState:=bolState); // get global/base defined cmds/states

IF (getCmdState='') THEN // global not defined get local
	// get string cmd/state string information in runtime
	IF (bolState=FALSE) THEN
		CASE intCmdState OF
			PBC_CmdState.cCMD_SINGLE: 
				getCmdState := 'cCMD_SINGLE';
			PBC_CmdState.cCMD_STANDBY: 
				getCmdState := 'cCMD_STANDBY';
		END_CASE;
	ELSE
		// States's
		CASE intCmdState OF
			PBC_CmdState.cSTA_STANDBYBusy: 
				getCmdState := 'cSTA_STANDBYBusy';
			PBC_CmdState.cSTA_STANDBY: 
				getCmdState := 'cSTA_STANDBY';
			PBC_CmdState.cSTA_EjectBusy: 
				getCmdState := 'cSTA_EjectBusy';
			PBC_CmdState.cSTA_EjectCheck: 
				getCmdState := 'cSTA_EjectCheck';
			PBC_CmdState.cSTA_PositionPaperBusy: 
				getCmdState := 'cSTA_PositionPaperBusy';
			PBC_CmdState.cSTA_RUNEmpty: 
				getCmdState := 'cSTA_RUNEmpty';
			PBC_CmdState.cSUB_WAITPAPER: 
				getCmdState := 'WAITPAPER';
			PBC_CmdState.cSUB_EJECTSTARTbusy: 
				getCmdState := 'EJECTSTARTbusy';
			PBC_CmdState.cSUB_EJECTbusy: 
				getCmdState := 'EJECTbusy';

			PBC_CmdState.cSUB_EJECTSTOPbusy: 
				getCmdState := 'EJECTSTOPbusy';
			PBC_CmdState.cSUB_EVALUATEEJECT: 
				getCmdState := 'EVALUATEEJECT';
			PBC_CmdState.cSUB_POSITIONbusy: 
				getCmdState := 'POSITIONbusy';

			PBC_CmdState.cSUB_POSITIONSTARTbusy: 
				getCmdState := 'POSITIONSTARTbusy';
			PBC_CmdState.cSUB_POSITIONSTOPbusy: 
				getCmdState := 'POSITIONSTOPbusy';
			PBC_CmdState.cSUB_READYEJECT: 
				getCmdState := 'READYEJECT';
			PBC_CmdState.cSUB_WAITPAPERGONETABLE: 
				getCmdState := 'WAITPAPERGONETABLE';
			PBC_CmdState.cSUB_POSITIONRETRYDELAY: 
				getCmdState := 'POSITIONRETRYDELAY';
			PBC_CmdState.cSUB_POSITIONRETRYSTOP: 
				getCmdState := 'POSITIONRETRYSTOP';
		END_CASE;
	END_IF
END_IF
END_METHOD

{attribute 'object_name' := 'getCtrlSIf'}
METHOD getCtrlSIf : POINTER TO T_Ctrl_SIf_PBC
getCtrlSIf := ADR(SIf);
END_METHOD

{attribute 'object_name' := 'IoInBridge'}
METHOD PROTECTED IoInBridge : BOOL
// digitale and analoge inputs read from hardware or forcing
SIf.In.bolCapacityReached.map			:= THIS^.In_bolCapacityReached				;
SIf.In.bolPaperAvailableEntry.map		:= THIS^.In_bolPaperAvailableEntry	;
SIf.In.bolPaperAvailableExit.map		:= THIS^.In_bolPaperAvailableExit		;
SIf.In.bolDoublePaperDetection.map		:= NOT THIS^.In_bolDoublePaperDetection		;
SIf.In.bolTurnTableMiddleSensor.map		:= NOT THIS^.In_bolTurnTableMiddleSensor		;
SIf.In.bolAirPressorOk.map				:= THIS^.In_bolAirPressorOk		;

IF (CIf.SwCfg.bolSimulation = FALSE) THEN
	BASE_PLC.getInBol(CIf.Job.bolIoForce,ADR(SIf.In.bolCapacityReached));
	BASE_PLC.getInBol(CIf.Job.bolIoForce,ADR(SIf.In.bolPaperAvailableEntry));
	BASE_PLC.getInBol(CIf.Job.bolIoForce,ADR(SIf.In.bolPaperAvailableExit));
	BASE_PLC.getInBolDebounced(CIf.Job.bolIoForce,me.FUBInfo.udiSample_ms, SIf.Par.udiDoublePaperDebounceTime_ms, ADR(SIf.In.bolDoublePaperDetection));
	BASE_PLC.getInBol(CIf.Job.bolIoForce,ADR(SIf.In.bolTurnTableMiddleSensor));
	BASE_PLC.getInBol(CIf.Job.bolIoForce,ADR(SIf.In.bolAirPressorOk));
ELSE
;	//simulation of global IO
END_IF
END_METHOD

{attribute 'object_name' := 'IoOutBridge'}
METHOD PROTECTED IoOutBridge : BOOL
VAR
	bolSwitchValvesOff: BOOL;
END_VAR
// digitale and analoge inputs read from hardware or forcing
IF (CIf.SwCfg.bolSimulation = FALSE) THEN
	setOutBol(CIf.Job.bolIoForce ,ADR(SIf.Out.bolAirOn));
	THIS^.Out_bolAirOn := SIf.Out.bolAirOn.map;
END_IF
END_METHOD

PROPERTY PaperHight : UINT
GET
PaperHight := m_uinPaperHight_mm;
END_GET
SET
m_uinPaperHight_mm := PaperHight;
END_SET
END_PROPERTY

PROPERTY PaperWidth : UINT
GET
PaperWidth := m_uinPaperWidth_mm;
END_GET
SET
m_uinPaperWidth_mm := PaperWidth;
END_SET
END_PROPERTY

{attribute 'object_name' := 'sta_EjectBusy'}
METHOD PROTECTED sta_EjectBusy : BOOL
// state implemetation
//--------------------------------------------------------------------------------------
// Entry action
IF (me.StateMachine.intState<>me.StateMachine.intStateLastCycle) THEN
	me.StateMachine.intStateLastCycle := me.StateMachine.intState;
	pDeStackerCIf^.Job.intACmd := BASE_PLC.cCMD_RUN;

	SIf.Cur.bolPaperBeforeEjectAvailable := SIf.In.bolPaperAvailableEntry.intern;
	SIf.Cur.uinPaperToPaperTime_ms := UDINT_TO_UINT((m_uinPaperHight_mm + 100) * 1000 / p_fbDeStacker^.CtrlSIf^.Par.rBeltParam.uinBeltSpeed);

// - SIMULATION ------------------------------------------------------------------------------------------- 		
	IF CIf.SwCfg.bolSimulation THEN
		fbSimulationTimer.IN := FALSE;
		fbSimulationTimer.PT := UDINT_TO_TIME(SIf.Par.udiSimPaperTransportTime);
		fbSimulationTimer(); // set time/reset timer
		fbSimulationTimer.IN := TRUE; // start timer
	END_IF
// -------------------------------------------------------------------------------------------- 		
END_IF


//--------------------------------------------------------------------------------------
// Cyclic action
IF (me.StateMachine.intState=me.StateMachine.intStateLastCycle) THEN

// - SIMULATION ------------------------------------------------------------------------------------------- 		
	IF (CIf.SwCfg.bolSimulation) THEN
		fbSimulationTimer(); // simulation time

		IF (fbSimulationTimer.Q) THEN
			SIf.In.bolPaperAvailableExit.intern := FALSE;
		END_IF
	END_IF
// -------------------------------------------------------------------------------------------- 		

	IF NOT SIf.In.bolPaperAvailableExit.intern THEN
		IF SIf.Cur.uinPaperToEjectParameter > 0 THEN
			SIf.Cur.uinPaperToEjectCount := SIf.Cur.uinPaperToEjectCount - 1;
		END_IF

		IF SIf.Cur.bolPaperBeforeEjectAvailable THEN
			me.StateMachine.intStateNext := PBC_CmdState.cSTA_PositionPaperBusy;
		ELSE
			me.StateMachine.intStateNext := PBC_CmdState.cSTA_EjectCheck;
			pfbAlarmCtrl^.setAlarm(CIf.Info.intCtrlId,INT_TO_UINT(E_ALM_PBC.BufferEmpty),0,ADR(SIf.Alm),E_AlmState.RST,CIf.Job.eMe_ActivAlmClass);
		END_IF
	END_IF

	IF (me.StateMachine.udiTimeInState_ms > SIf.Cur.uinPaperToPaperTime_ms) THEN
		pfbAlarmCtrl^.setAlarm(CIf.Info.intCtrlId,INT_TO_UINT(E_ALM_PBC.PaperTransport),0,ADR(SIf.Alm),E_AlmState.RST,CIf.Job.eMe_ActivAlmClass);
		me.StateMachine.intStateNext := Base_PLC.cSTA_ERROR;	
	END_IF
END_IF


//--------------------------------------------------------------------------------------
// Exit action
IF (me.StateMachine.intState<>me.StateMachine.intStateNext) THEN
	;
END_IF
END_METHOD

{attribute 'object_name' := 'sta_EjectCheck'}
METHOD PROTECTED sta_EjectCheck : BOOL
// state implemetation
//--------------------------------------------------------------------------------------
// Entry action
	IF (me.StateMachine.intState<>me.StateMachine.intStateLastCycle) THEN
		me.StateMachine.intStateLastCycle := me.StateMachine.intState;
//		SIf.Cur.bolPaperBeforeEjectAvailable := SIf.In.bolPaperAvailableEntry.intern;
	END_IF


//--------------------------------------------------------------------------------------
// Cyclic action
	IF (me.StateMachine.intState=me.StateMachine.intStateLastCycle) THEN
			
		// Eject next paper if there are still paper to edject or endless ejection
		IF (SIf.Cur.uinPaperToEjectCount > 0) OR (SIf.Cur.uinPaperToEjectParameter = 0) THEN
			// Make a delay from sheet to sheet if it is not the first sheet
			IF   (SIf.Cur.uinSheetToSheetTime > SIf.Par.udiSheetToSheetTime) 
			  OR (SIf.Cur.uinPaperToEjectCount = SIf.Cur.uinPaperToEjectParameter) THEN
				IF SIf.In.bolPaperAvailableExit.intern THEN
					SIf.Cur.uinSheetToSheetTime := 0;
					me.StateMachine.intStateNext := PBC_CmdState.cSTA_EjectBusy;
				ELSE
					IF SIf.In.bolPaperAvailableEntry.intern THEN
						me.StateMachine.intStateNext := PBC_CmdState.cSTA_PositionPaperBusy;
					END_IF
				END_IF
			END_IF
		ELSE
			me.StateMachine.intStateNext := PBC_CmdState.cSTA_STANDBYBusy;
		END_IF

		CASE me.intCmd OF
			BASE_PLC.cCMD_STOP:
				me.StateMachine.intStateNext := PBC_CmdState.cSTA_STANDBYBusy;
			PBC_CmdState.cCMD_STANDBY:
				me.StateMachine.intStateNext := PBC_CmdState.cSTA_STANDBYBusy;
		END_CASE
	END_IF


//--------------------------------------------------------------------------------------
// Exit action
	IF (me.StateMachine.intState<>me.StateMachine.intStateNext) THEN
		;
	END_IF
END_METHOD

{attribute 'object_name' := 'sta_ERROR'}
METHOD PROTECTED sta_ERROR : BOOL
// state implemetation
//--------------------------------------------------------------------------------------
// Entry action
	IF (me.StateMachine.intState<>me.StateMachine.intStateLastCycle) THEN
		me.StateMachine.intStateHistory := me.StateMachine.intStateLastCycle; // -> possibillity to go back to state before error
		me.StateMachine.intStateLastCycle := me.StateMachine.intState;
		pDeStackerCIf^.Job.intACmd 	:= BASE_PLC.cCMD_STOP;
		//pBeltCIf^.Job.intACmd 		:= BASE_PLC.cCMD_STOP;
	END_IF


//--------------------------------------------------------------------------------------
// Cyclic action
	IF (me.StateMachine.intState=me.StateMachine.intStateLastCycle) THEN
		
		;
		
		
		// State Change Condition
		IF (CIf.Job.bolAlmReset = TRUE) THEN
			me.StateMachine.intStateNext := cSTA_ERRORQuit;
		END_IF
	END_IF




//--------------------------------------------------------------------------------------
// Exit action
	IF (me.StateMachine.intState<>me.StateMachine.intStateNext) THEN
		;
	END_IF
END_METHOD

{attribute 'object_name' := 'sta_ERRORQuit'}
METHOD PROTECTED sta_ERRORQuit : BOOL
// state implemetation
//--------------------------------------------------------------------------------------
// Entry action
	IF (me.StateMachine.intState<>me.StateMachine.intStateLastCycle) THEN
		me.StateMachine.intStateLastCycle := me.StateMachine.intState;
		
	END_IF


//--------------------------------------------------------------------------------------
// Cyclic action
	IF (me.StateMachine.intState=me.StateMachine.intStateLastCycle) THEN
		
		;
		// evtl. wait time if reset of device is necessary and then decide to go to states or ERROR state
		IF (CIf.Job.bolAlmReset = TRUE) THEN
			CIf.Job.eMe_ActivAlmClass := E_AlmClass.NONE; // reset feedback channel for parent
			CIf.Job.bolAlmReset := FALSE;
		END_IF
		
		// State Change Condition
		IF (CIf.Job.bolAlmReset = FALSE) THEN
			IF (me.StateMachine.intStateHistory<=BASE_PLC.cSTA_PON) THEN
				me.StateMachine.intStateNext := BASE_PLC.cSTA_PONBusy;
			END_IF;

			CASE me.intCmd OF
				BASE_PLC.cCMD_OFF:
					me.StateMachine.intStateNext := BASE_PLC.cSTA_OFFBusy;
				PBC_CmdState.cCMD_STANDBY:
					me.StateMachine.intStateNext := PBC_CmdState.cSTA_STANDBYBusy;
				PBC_CmdState.cCMD_SINGLE,
				BASE_PLC.cCMD_RUN:
					me.StateMachine.intStateNext := BASE_PLC.cSTA_RUNBusy;
			ELSE
				CASE me.StateMachine.intStateHistory OF
					PBC_CmdState.cSTA_STANDBY:
						me.StateMachine.intStateNext := PBC_CmdState.cSTA_STANDBYBusy;
					BASE_PLC.cSTA_RUN:
						me.StateMachine.intStateNext := BASE_PLC.cSTA_RUNBusy;
				END_CASE
			END_CASE
		END_IF
	END_IF




//--------------------------------------------------------------------------------------
// Exit action
	IF (me.StateMachine.intState<>me.StateMachine.intStateNext) THEN
		;
	END_IF
END_METHOD

{attribute 'object_name' := 'sta_OFF'}
METHOD PROTECTED sta_OFF : BOOL
// state implemetation
//--------------------------------------------------------------------------------------
// Entry action
	IF (me.StateMachine.intState<>me.StateMachine.intStateLastCycle) THEN
		me.StateMachine.intStateLastCycle := me.StateMachine.intState;

	END_IF


//--------------------------------------------------------------------------------------
// Cyclic action
	IF (me.StateMachine.intState=me.StateMachine.intStateLastCycle) THEN
		CASE me.intCmd OF
			BASE_PLC.cCMD_RUN : 
				me.StateMachine.intStateNext := PBC_CmdState.cSTA_STANDBYBusy;
			PBC_CmdState.cCMD_STANDBY : 
				me.StateMachine.intStateNext := PBC_CmdState.cSTA_STANDBYBusy;
		END_CASE
	END_IF


//--------------------------------------------------------------------------------------
// Exit action
	IF (me.StateMachine.intState<>me.StateMachine.intStateNext) THEN
		;
	END_IF
END_METHOD

{attribute 'object_name' := 'sta_OFFBusy'}
METHOD PROTECTED sta_OFFBusy : BOOL
// state implemetation
//--------------------------------------------------------------------------------------
// Entry action
	IF (me.StateMachine.intState<>me.StateMachine.intStateLastCycle) THEN
		me.StateMachine.intStateLastCycle := me.StateMachine.intState;
		
		SIf.Out.bolAirOn.intern := FALSE;
		
		pDeStackerCIf^.Job.intACmd := BASE_PLC.cCMD_OFF;
		pBeltCIf^.Job.intACmd := BASE_PLC.cCMD_OFF;
	END_IF


//--------------------------------------------------------------------------------------
// Cyclic action
	IF (me.StateMachine.intState=me.StateMachine.intStateLastCycle) THEN
		IF (pDeStackerCIf^.Job.intState = BASE_PLC.cSTA_OFF)
		  AND (pBeltCIf^.Job.intState = BASE_PLC.cSTA_OFF) 
		  AND (NOT SIf.In.bolAirPressorOk.intern OR (NOT SIf.Cfg.bolGranulatAirPressureUnitAvailable))  THEN
			me.StateMachine.intStateNext := BASE_PLC.cSTA_OFF;
		END_IF
	END_IF


//--------------------------------------------------------------------------------------
// Exit action
	IF (me.StateMachine.intState<>me.StateMachine.intStateNext) THEN
		;
	END_IF
END_METHOD

{attribute 'object_name' := 'sta_PON'}
METHOD PROTECTED sta_PON : BOOL
// state implemetation
//--------------------------------------------------------------------------------------
// Entry action
	IF (me.StateMachine.intState<>me.StateMachine.intStateLastCycle) THEN
		me.StateMachine.intStateLastCycle := me.StateMachine.intState;
		
	END_IF


//--------------------------------------------------------------------------------------
// Cyclic action
	IF (me.StateMachine.intState=me.StateMachine.intStateLastCycle) THEN
		;
	END_IF




//--------------------------------------------------------------------------------------
// Exit action
	IF (me.StateMachine.intState<>me.StateMachine.intStateNext) THEN
		;
	END_IF
END_METHOD

{attribute 'object_name' := 'sta_PositionPaperBusy'}
METHOD PROTECTED sta_PositionPaperBusy : BOOL
(*
// state implemetation
//--------------------------------------------------------------------------------------
// Entry action
IF (me.StateMachine.intState<>me.StateMachine.intStateLastCycle) THEN
	me.StateMachine.intStateLastCycle := me.StateMachine.intState;
	CIf.Job.intACmd := BASE_PLC.cCMD_DONE;
	CIf.Job.intMCmd := BASE_PLC.cCMD_DONE;
	
	IF NOT SIf.In.bolPaperAvailableExit.intern THEN
		pDeStackerCIf^.Job.intACmd := BASE_PLC.cCMD_RUN;
	END_IF

	me.SubStateMachine.intState := PBC_CmdState.cSUB_WAITPAPER;
	me.SubStateMachine.intStateNext := PBC_CmdState.cSUB_WAITPAPER;

// - SIMULATION ------------------------------------------------------------------------------------------- 		
	IF CIf.SwCfg.bolSimulation THEN
		fbSimulationTimer.IN := FALSE;
		fbSimulationTimer.PT := UDINT_TO_TIME(SIf.Par.udiSimPaperToPaperTransportTime);
		fbSimulationTimer(); // set time/reset timer
		fbSimulationTimer.IN := TRUE; // start timer
	END_IF
// -------------------------------------------------------------------------------------------- 		
END_IF


//-------------------------------------------------------------------------------------- 
// Cyclic action
IF (me.StateMachine.intState=me.StateMachine.intStateLastCycle) THEN
// - SIMULATION ------------------------------------------------------------------------------------------- 		
	IF (CIf.SwCfg.bolSimulation) THEN
		fbSimulationTimer(); // simulation time

		IF (fbSimulationTimer.Q) THEN
			SIf.In.bolPaperAvailableExit.intern := TRUE;
		END_IF
	END_IF
// -------------------------------------------------------------------------------------------- 		

	CASE me.SubStateMachine.intState OF
		PBC_CmdState.cSUB_STARTDRIVE:
			pDeStackerCIf^.Job.intACmd := BASE_PLC.cCMD_RUN;
			me.SubStateMachine.intStateNext := PBC_CmdState.cSUB_WAITPAPER;
			
		PBC_CmdState.cSUB_WAITPAPER:
			IF SIf.In.bolPaperAvailableExit.intern THEN
				pDeStackerCIf^.Job.intACmd := BASE_PLC.cCMD_STOP;
				me.SubStateMachine.intStateNext := PBC_CmdState.cSUB_WAITSTOP;
			END_IF

			IF (me.SubStateMachine.udiTimeInState_ms > SIf.Par.udiPaperTransportTime) THEN
				IF SIf.Cur.bolPaperBeforeEjectAvailable THEN
					g_fbAlm_Man.setAlarm(CIf.Info.intCtrlId,INT_TO_UINT(E_ALM_PBC.PaperTransport),0,ADR(SIf.Alm),E_AlmState.RST,CIf.Job.eMe_ActivAlmClass);
					me.StateMachine.intStateNext := Base_PLC.cSTA_ERROR;	
				ELSE
					pDeStackerCIf^.Job.intACmd := BASE_PLC.cCMD_STOP;
					me.StateMachine.intStateNext := PBC_CmdState.cSTA_STANDBYBusy;
				END_IF
			END_IF
			
		PBC_CmdState.cSUB_WAITSTOP:
			IF pDeStackerCIf^.Job.intState = BASE_PLC.cSTA_STOP THEN
				me.StateMachine.intStateNext := PBC_CmdState.cSTA_EjectCheck;
			END_IF			
	END_CASE
END_IF


//--------------------------------------------------------------------------------------
// Exit action
IF (me.StateMachine.intState<>me.StateMachine.intStateNext) THEN
	me.SubStateMachine.intState := BASE_PLC.cSTA_INITIALIZED;
	me.SubStateMachine.intStateNext := BASE_PLC.cSTA_INITIALIZED;
END_IF
*)
END_METHOD

{attribute 'object_name' := 'sta_RUN'}
METHOD PROTECTED sta_RUN : BOOL
VAR
	pItem: POINTER TO T_IdBase_DCH;
END_VAR
// state implemetation
//--------------------------------------------------------------------------------------
// Entry action
IF (me.StateMachine.intState<>me.StateMachine.intStateLastCycle) THEN
	me.StateMachine.intStateLastCycle := me.StateMachine.intState;
	
	IF (me.intCmd = BASE_PLC.cCMD_RUN) OR (me.intCmd = PBC_CmdState.cCMD_SINGLE) THEN
		CIf.Job.intACmd := BASE_PLC.cCMD_DONE;
		CIf.Job.intMCmd := BASE_PLC.cCMD_DONE;
	END_IF
	
	SIf.Cur.uinSheetToSheetTime := 0;
	m_intRetry := 0;
	
	IF CIf.SwCfg.bolSimulation THEN
		SIf.In.bolPaperAvailableEntry.intern := TRUE;
		SIf.In.bolDoublePaperDetection.intern := FALSE;	
		SIf.In.bolPaperAvailableExit.intern := TRUE;	
		SIf.In.bolCapacityReached.intern := TRUE;
	END_IF

	me.SubStateMachine.intState 	:= PBC_CmdState.cSUB_POSITIONSTARTbusy;
	me.SubStateMachine.intStateNext := PBC_CmdState.cSUB_POSITIONSTARTbusy;
END_IF


//--------------------------------------------------------------------------------------
// Cyclic action
IF (me.StateMachine.intState=me.StateMachine.intStateLastCycle) THEN
	IF (SIf.In.bolDoublePaperDetection.intern) THEN
		pfbAlarmCtrl^.setAlarm(CIf.Info.intCtrlId,INT_TO_UINT(E_ALM_PBC.DoublePaper),0,ADR(SIf.Alm),E_AlmState.RST,CIf.Job.eMe_ActivAlmClass);
		
		IF SIf.Par.bolEnableDoublePaperDetection THEN
			me.StateMachine.intStateNext := Base_PLC.cSTA_ERROR;
		END_IF
	ELSE	
		CASE me.SubStateMachine.intState OF
			// substate Wait paper - wait for the next paper if the buffer was empty
			// ------------------------------------------------------------------------
			PBC_CmdState.cSUB_WAITPAPER:
				IF NOT SIf.In.bolPaperAvailableExit.intern THEN
					IF SIf.In.bolCapacityReached.intern THEN
						me.SubStateMachine.intStateNext := PBC_CmdState.cSUB_POSITIONSTARTbusy;
					END_IF
				END_IF
				
			// substate Wait paper - wait for the next paper if the buffer was empty
			// ------------------------------------------------------------------------
			PBC_CmdState.cSUB_POSITIONSTARTbusy:
				IF NOT SIf.In.bolPaperAvailableExit.intern THEN
					SIf.Cur.bolPaperBeforeEjectAvailable := SIf.In.bolCapacityReached.intern;
					pDeStackerCIf^.Job.intACmd := BASE_PLC.cCMD_RUN;
					me.SubStateMachine.intStateNext := PBC_CmdState.cSUB_POSITIONbusy;
				ELSE
					me.SubStateMachine.intStateNext := cSUB_EVALUATEEJECT;
				END_IF
	
			// substate Wait paper - wait for the next paper if the buffer was empty
			// ------------------------------------------------------------------------
			PBC_CmdState.cSUB_POSITIONbusy:
				IF me.SubStateMachine.udiTimeInState_ms <= SIf.Par.udiPaperTransportTime THEN
					IF SIf.In.bolPaperAvailableExit.intern THEN
						m_intRetry := 0;
						pDeStackerCIf^.Job.intACmd := BASE_PLC.cCMD_STOP;
						me.SubStateMachine.intStateNext := PBC_CmdState.cSUB_POSITIONSTOPbusy;
					END_IF
				ELSE
					IF SIf.Cur.bolPaperBeforeEjectAvailable THEN
						IF DINT_TO_UDINT(m_intRetry) < SIf.Par.udiPaperInjectRetries THEN
							pDeStackerCIf^.Job.intACmd := BASE_PLC.cCMD_STOP;
							m_intRetry := m_intRetry + 1;
							pfbAlarmCtrl^.setAlarm(CIf.Info.intCtrlId,INT_TO_UINT(E_ALM_PBC.PaperInjectRetry),m_intRetry,ADR(SIf.Alm),E_AlmState.RST,CIf.Job.eMe_ActivAlmClass);
							me.SubStateMachine.intStateNext := PBC_CmdState.cSUB_POSITIONRETRYSTOP;	
						ELSE
							m_intRetry := 0;
							pfbAlarmCtrl^.setAlarm(CIf.Info.intCtrlId,INT_TO_UINT(E_ALM_PBC.PaperInject),0,ADR(SIf.Alm),E_AlmState.RST,CIf.Job.eMe_ActivAlmClass);
							me.StateMachine.intStateNext := Base_PLC.cSTA_ERROR;	
						END_IF
					ELSE
						m_intRetry := 0;
						pDeStackerCIf^.Job.intACmd := BASE_PLC.cCMD_STOP;
						me.SubStateMachine.intStateNext := PBC_CmdState.cSUB_POSITIONSTOPbusy;
					END_IF 
				END_IF

				// Simulation
				IF CIf.SwCfg.bolSimulation THEN
					IF (me.SubStateMachine.udiTimeInState_ms > SIf.Par.udiSimPaperTransportTime) AND NOT SIf.In.bolPaperAvailableExit.intern THEN
						SIf.In.bolPaperAvailableExit.intern := TRUE;	
					END_IF
				END_IF
				// -----------------------------------
	
			// Wait that the moto stops
			// ------------------------------------------------------------------------
			PBC_CmdState.cSUB_POSITIONRETRYSTOP:
				IF pDeStackerCIf^.Job.intState = BASE_PLC.cSTA_STOP THEN
					me.SubStateMachine.intStateNext := PBC_CmdState.cSUB_POSITIONRETRYDELAY;
				END_IF

			// Stop the motor and way for x ms
			// ------------------------------------------------------------------------
			PBC_CmdState.cSUB_POSITIONRETRYDELAY:
				IF me.SubStateMachine.udiTimeInState_ms > SIf.Par.udiPaperInjectRetryPauseTime_ms THEN
					me.SubStateMachine.intStateNext := PBC_CmdState.cSUB_POSITIONSTARTbusy;
				END_IF

			// substate Wait paper - wait for the next paper if the buffer was empty
			// ------------------------------------------------------------------------
			PBC_CmdState.cSUB_POSITIONSTOPbusy:
				IF pDeStackerCIf^.Job.intState = BASE_PLC.cSTA_STOP THEN
					IF SIf.In.bolPaperAvailableExit.intern THEN
						me.SubStateMachine.intStateNext := PBC_CmdState.cSUB_EVALUATEEJECT;
					ELSE
						me.SubStateMachine.intStateNext := PBC_CmdState.cSUB_WAITPAPER;
					END_IF
				END_IF

			// substate Wait paper - wait for the next paper if the buffer was empty
			// ------------------------------------------------------------------------
			PBC_CmdState.cSUB_EVALUATEEJECT:
				// Eject next paper if there are still paper to edject or endless ejection
				IF (SIf.Cur.uinPaperToEjectCount > 0) OR (SIf.Cur.uinPaperToEjectParameter = 0) OR SIf.Par.bolAutomaticMode THEN
					// Make a delay from sheet to sheet if it is not the first sheet
					IF   (SIf.Cur.uinSheetToSheetTime > SIf.Par.udiSheetToSheetTime) 
					  OR (SIf.Cur.uinPaperToEjectCount = SIf.Cur.uinPaperToEjectParameter) THEN
						SIf.Cur.uinSheetToSheetTime := 0;
	
						IF SIf.In.bolPaperAvailableExit.intern THEN
							me.SubStateMachine.intStateNext := PBC_CmdState.cSUB_EJECTSTARTbusy;
						ELSE
							me.SubStateMachine.intStateNext := PBC_CmdState.cSUB_WAITPAPER;
						END_IF
					END_IF
				ELSE
					me.StateMachine.intStateNext := PBC_CmdState.cSTA_STANDBYBusy;
				END_IF
	
			// substate Wait paper - wait for the next paper if the buffer was empty
			// ------------------------------------------------------------------------
			PBC_CmdState.cSUB_EJECTSTARTbusy:
				pDeStackerCIf^.Job.intACmd := BASE_PLC.cCMD_RUN;
				SIf.Cur.uinPaperToPaperTime_ms := UDINT_TO_UINT((m_uinPaperHight_mm + 100) * 1000 / p_fbDeStacker^.CtrlSIf^.Par.rBeltParam.uinBeltSpeed);
				SIf.Par.udiSimPaperToPaperTransportTime := SIf.Cur.uinPaperToPaperTime_ms / 3; 
				me.SubStateMachine.intStateNext := PBC_CmdState.cSUB_EJECTbusy;
	
			// substate Wait paper - wait for the next paper if the buffer was empty
			// ------------------------------------------------------------------------
			PBC_CmdState.cSUB_EJECTbusy:
				IF NOT SIf.In.bolPaperAvailableExit.intern AND NOT SIf.Cfg.bolUseTurnTableSensorForEject THEN
					pDeStackerCIf^.Job.intACmd := BASE_PLC.cCMD_STOP;
					me.SubStateMachine.intStateNext := PBC_CmdState.cSUB_EJECTSTOPbusy;
				END_IF
	
				IF SIf.In.bolTurnTableMiddleSensor.intern AND SIf.Cfg.bolUseTurnTableSensorForEject THEN
					pDeStackerCIf^.Job.intACmd := BASE_PLC.cCMD_STOP;
					me.SubStateMachine.intStateNext := PBC_CmdState.cSUB_WAITPAPERGONETABLE;
				END_IF
				
				IF (me.SubStateMachine.udiTimeInState_ms > SIf.Cur.uinPaperToPaperTime_ms) THEN
					pfbAlarmCtrl^.setAlarm(CIf.Info.intCtrlId,INT_TO_UINT(E_ALM_PBC.PaperTransport),0,ADR(SIf.Alm),E_AlmState.RST,CIf.Job.eMe_ActivAlmClass);
					me.StateMachine.intStateNext := Base_PLC.cSTA_ERROR;	
				END_IF

				// Simulation
				IF CIf.SwCfg.bolSimulation THEN
					IF (me.SubStateMachine.udiTimeInState_ms > SIf.Par.udiSimPaperToPaperTransportTime) THEN
						IF SIf.Cfg.bolUseTurnTableSensorForEject THEN
							SIf.In.bolTurnTableMiddleSensor.intern := TRUE;
						ELSE
							SIf.In.bolPaperAvailableExit.intern := FALSE;	
						END_IF	
					END_IF
				END_IF
				// -----------------------------------
	
			// substate Wait Paper Gone Table - Wait until the paper is gone from the turn table
			// ------------------------------------------------------------------------
			PBC_CmdState.cSUB_WAITPAPERGONETABLE:
				IF NOT SIf.In.bolTurnTableMiddleSensor.intern THEN
					me.SubStateMachine.intStateNext := PBC_CmdState.cSUB_EJECTSTOPbusy;
				END_IF

				// Simulation
				IF CIf.SwCfg.bolSimulation THEN
					IF (me.SubStateMachine.udiTimeInState_ms > SIf.Par.udiSimPaperToPaperTransportTime) THEN
						SIf.In.bolTurnTableMiddleSensor.intern := FALSE;
					END_IF
				END_IF
				// -----------------------------------

	
			// substate Wait paper - wait for the next paper if the buffer was empty
			// ------------------------------------------------------------------------
			PBC_CmdState.cSUB_EJECTSTOPbusy:
				IF pDeStackerCIf^.Job.intState = BASE_PLC.cSTA_STOP THEN
					IF SIf.Cur.uinPaperToEjectCount > 0 THEN
						SIf.Cur.uinPaperToEjectCount := SIf.Cur.uinPaperToEjectCount - 1;
					END_IF
	
					me.SubStateMachine.intStateNext := PBC_CmdState.cSUB_POSITIONSTARTbusy;
				END_IF
		END_CASE
	END_IF
	
	CASE me.SubStateMachine.intState OF
		PBC_CmdState.cSUB_WAITPAPER,
		PBC_CmdState.cSUB_EVALUATEEJECT:
			CASE me.intCmd OF
				PBC_CmdState.cCMD_STANDBY:
					me.StateMachine.intStateNext := PBC_CmdState.cSTA_STANDBYBusy;
				BASE_PLC.cCMD_STOP:
					me.StateMachine.intStateNext := BASE_PLC.cSTA_STOPBusy;
			END_CASE
	END_CASE
	
	SIf.Cur.uinSheetToSheetTime := UDINT_TO_UINT(SIf.Cur.uinSheetToSheetTime + me.FUBInfo.udiSample_ms);
END_IF


//--------------------------------------------------------------------------------------
// Exit action
IF (me.StateMachine.intState<>me.StateMachine.intStateNext) THEN
	me.SubStateMachine.intState 	:= BASE_PLC.cSTA_INITIALIZED;
	me.SubStateMachine.intStateNext := BASE_PLC.cSTA_INITIALIZED;
END_IF
END_METHOD

